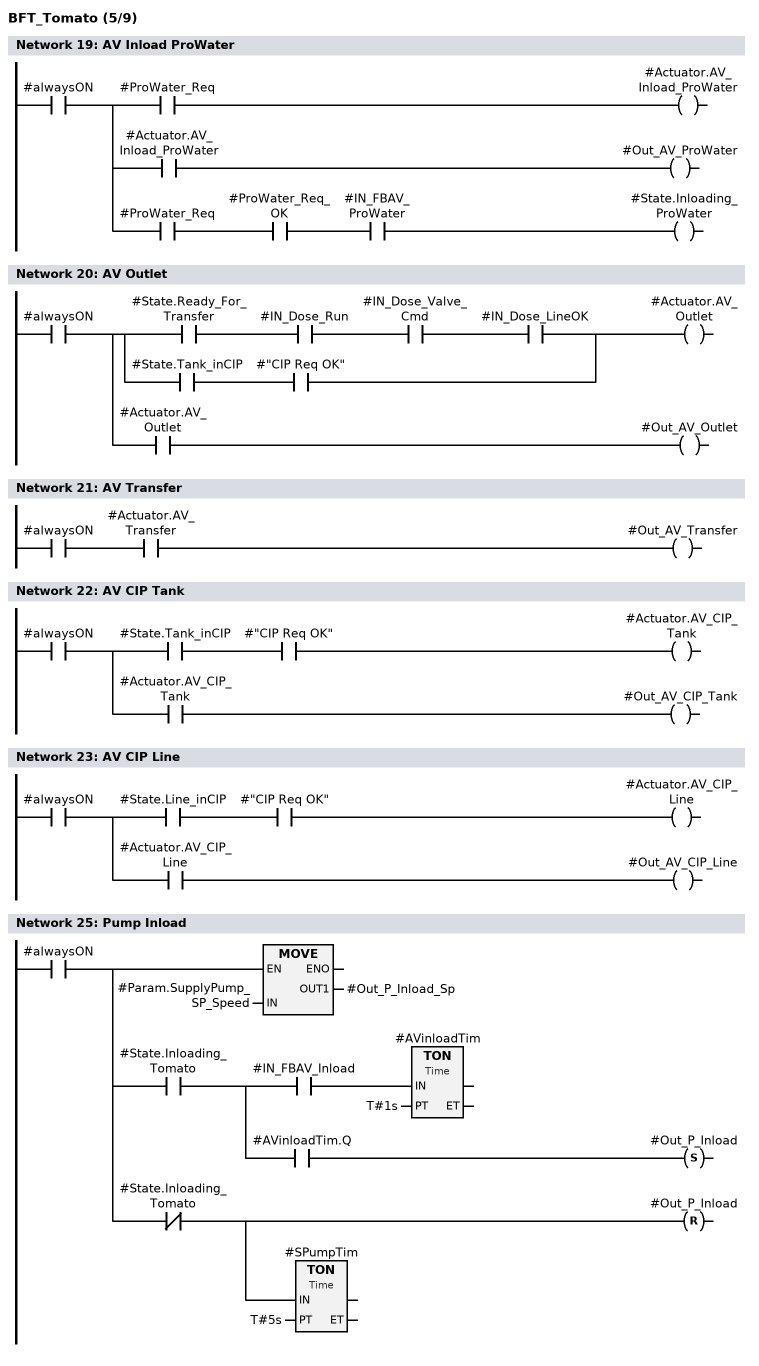
   RUNG wire#powerrail
      Contact( #alwaysON )
      wire#w1
      Contact( #ProWater_Req )
      Coil( #Actuator.AV_Inload_ProWater )
   END_RUNG
   RUNG wire#w1
      Contact( #Actuator.AV_Inload_ProWater )
      Coil( #Out_AV_ProWater )
   END_RUNG
   RUNG wire#w1
      Contact( #ProWater_Req )
      Contact( #ProWater_Req_OK )
      Contact( #IN_FBAV_ProWater )
      Coil( #State.Inloading_ProWater )
   END_RUNG
   // the same network as SCL:
   #Actuator.AV_Inload_ProWater := #alwaysON AND #ProWater_Req;
   #Out_AV_ProWater := #alwaysON AND #Actuator.AV_Inload_ProWater;
   #State.Inloading_ProWater := #alwaysON AND #ProWater_Req AND #ProWater_Req_OK AND #IN_FBAV_ProWater;
END_REGION

REGION Network 20: AV Outlet
   RUNG wire#powerrail
      Contact( #alwaysON )
      wire#w1
      Contact( #State.Ready_For_Transfer )
      Contact( #IN_Dose_Run )
      Contact( #IN_Dose_Valve_Cmd )
      Contact( #IN_Dose_LineOK )
      wire#w2
      Coil( #Actuator.AV_Outlet )
   END_RUNG
   RUNG wire#w1
      Contact( #State.Tank_inCIP )
      Contact( #"CIP Req OK" )
   END_RUNG wire#w2
   RUNG wire#w1
      Contact( #Actuator.AV_Outlet )
      Coil( #Out_AV_Outlet )
   END_RUNG
   // the same network as SCL:
   #Actuator.AV_Outlet := #alwaysON AND ((#State.Ready_For_Transfer AND #IN_Dose_Run AND #IN_Dose_Valve_Cmd AND #IN_Dose_LineOK) OR (#State.Tank_inCIP AND #"CIP Req OK"));
   #Out_AV_Outlet := #alwaysON AND #Actuator.AV_Outlet;
END_REGION

REGION Network 21: AV Transfer
   RUNG wire#powerrail
      Contact( #alwaysON )
      Contact( #Actuator.AV_Transfer )
      Coil( #Out_AV_Transfer )
   END_RUNG
   // the same network as SCL:
   #Out_AV_Transfer := #alwaysON AND #Actuator.AV_Transfer;
END_REGION

REGION Network 22: AV CIP Tank
   RUNG wire#powerrail
      Contact( #alwaysON )
      wire#w1
      Contact( #State.Tank_inCIP )
      Contact( #"CIP Req OK" )
      Coil( #Actuator.AV_CIP_Tank )
   END_RUNG
   RUNG wire#w1
      Contact( #Actuator.AV_CIP_Tank )
      Coil( #Out_AV_CIP_Tank )
   END_RUNG
   // the same network as SCL:
   #Actuator.AV_CIP_Tank := #alwaysON AND #State.Tank_inCIP AND #"CIP Req OK";
   #Out_AV_CIP_Tank := #alwaysON AND #Actuator.AV_CIP_Tank;
END_REGION

REGION Network 23: AV CIP Line
   RUNG wire#powerrail
      Contact( #alwaysON )
      wire#w1
      Contact( #State.Line_inCIP )
      Contact( #"CIP Req OK" )
      Coil( #Actuator.AV_CIP_Line )
   END_RUNG
   RUNG wire#w1
      Contact( #Actuator.AV_CIP_Line )
      Coil( #Out_AV_CIP_Line )
   END_RUNG
   // the same network as SCL:
   #Actuator.AV_CIP_Line := #alwaysON AND #State.Line_inCIP AND #"CIP Req OK";
   #Out_AV_CIP_Line := #alwaysON AND #Actuator.AV_CIP_Line;
END_REGION

REGION Network 25: Pump Inload
   RUNG wire#powerrail
      Contact( #alwaysON )
      wire#w1
      Move(in := #Param.SupplyPump_SP_Speed, out1 => #Out_P_Inload_Sp)
   END_RUNG
   RUNG wire#w1
      Contact( #State.Inloading_Tomato )
      wire#w2
      Contact( #IN_FBAV_Inload )
      { S7_Templates := "time_type := Time" } #AVinloadTim.TON(pt := T#1s, et =>)
   END_RUNG
   RUNG wire#w2
      Contact( #AVinloadTim.Q )
      S_Coil( #Out_P_Inload )
   END_RUNG
   RUNG wire#w1
      I_Contact( #State.Inloading_Tomato )
      wire#w3
      R_Coil( #Out_P_Inload )
   END_RUNG
   RUNG wire#w3
      { S7_Templates := "time_type := Time" } #SPumpTim.TON(pt := T#5s, et =>)
   END_RUNG
   // the same network as SCL:
   IF #alwaysON THEN #Out_P_Inload_Sp := #Param.SupplyPump_SP_Speed; END_IF;
   #_w1 := #alwaysON AND #State.Inloading_Tomato;
   #AVinloadTim(IN := #_w1 AND #IN_FBAV_Inload, PT := T#1s);   // TON
   IF #_w1 AND #AVinloadTim.Q THEN #Out_P_Inload := TRUE; END_IF;
   #_w2 := #alwaysON AND NOT #State.Inloading_Tomato;
   IF #_w2 THEN #Out_P_Inload := FALSE; END_IF;
   #SPumpTim(IN := #_w2, PT := T#5s);   // TON
END_REGION

REGION Network 26: Pump Transfer
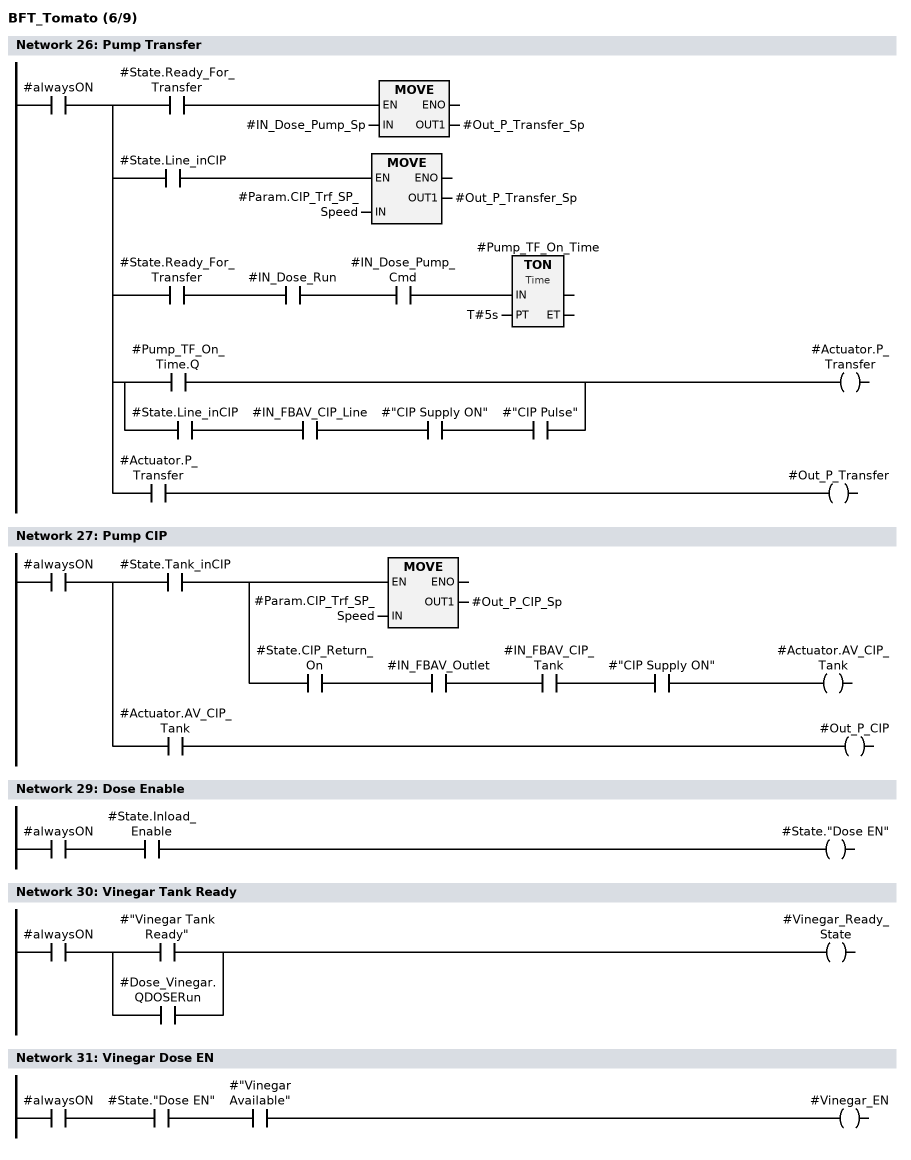
   RUNG wire#powerrail
      Contact( #alwaysON )
      wire#w1
      Contact( #State.Ready_For_Transfer )
      Move(in := #IN_Dose_Pump_Sp, out1 => #Out_P_Transfer_Sp)
   END_RUNG
   RUNG wire#w1
      Contact( #State.Line_inCIP )
      Move(in := #Param.CIP_Trf_SP_Speed, out1 => #Out_P_Transfer_Sp)
   END_RUNG
   RUNG wire#w1
      Contact( #State.Ready_For_Transfer )
      Contact( #IN_Dose_Run )
      Contact( #IN_Dose_Pump_Cmd )
      { S7_Templates := "time_type := Time" } #Pump_TF_On_Time.TON(pt := T#5s, et =>)
   END_RUNG
   RUNG wire#w1
      Contact( #Pump_TF_On_Time.Q )
      wire#w2
      Coil( #Actuator.P_Transfer )
   END_RUNG
   RUNG wire#w1
      Contact( #State.Line_inCIP )
      Contact( #IN_FBAV_CIP_Line )
      Contact( #"CIP Supply ON" )
      Contact( #"CIP Pulse" )
   END_RUNG wire#w2
   RUNG wire#w1
      Contact( #Actuator.P_Transfer )
      Coil( #Out_P_Transfer )
   END_RUNG
   // the same network as SCL:
   IF #alwaysON AND #State.Ready_For_Transfer THEN #Out_P_Transfer_Sp := #IN_Dose_Pump_Sp; END_IF;
   IF #alwaysON AND #State.Line_inCIP THEN #Out_P_Transfer_Sp := #Param.CIP_Trf_SP_Speed; END_IF;
   #Pump_TF_On_Time(IN := #alwaysON AND #State.Ready_For_Transfer AND #IN_Dose_Run AND #IN_Dose_Pump_Cmd,   // TON
                    PT := T#5s);
   #Actuator.P_Transfer := #alwaysON AND (#Pump_TF_On_Time.Q OR (#State.Line_inCIP AND #IN_FBAV_CIP_Line AND #"CIP Supply ON" AND #"CIP Pulse"));
   #Out_P_Transfer := #alwaysON AND #Actuator.P_Transfer;
END_REGION

REGION Network 27: Pump CIP
   RUNG wire#powerrail
      Contact( #alwaysON )
      wire#w1
      Contact( #State.Tank_inCIP )
      wire#w2
      Move(in := #Param.CIP_Trf_SP_Speed, out1 => #Out_P_CIP_Sp)
   END_RUNG
   RUNG wire#w2
      Contact( #State.CIP_Return_On )
      Contact( #IN_FBAV_Outlet )
      Contact( #IN_FBAV_CIP_Tank )
      Contact( #"CIP Supply ON" )
      Coil( #Actuator.AV_CIP_Tank )
   END_RUNG
   RUNG wire#w1
      Contact( #Actuator.AV_CIP_Tank )
      Coil( #Out_P_CIP )
   END_RUNG
   // the same network as SCL:
   #_w1 := #alwaysON AND #State.Tank_inCIP;
   IF #_w1 THEN #Out_P_CIP_Sp := #Param.CIP_Trf_SP_Speed; END_IF;
   #Actuator.AV_CIP_Tank := #_w1 AND #State.CIP_Return_On AND #IN_FBAV_Outlet AND #IN_FBAV_CIP_Tank AND #"CIP Supply ON";
   #Out_P_CIP := #alwaysON AND #Actuator.AV_CIP_Tank;
END_REGION

REGION Network 29: Dose Enable
   RUNG wire#powerrail
      Contact( #alwaysON )
      Contact( #State.Inload_Enable )
      Coil( #State."Dose EN" )
   END_RUNG
   // the same network as SCL:
   #State."Dose EN" := #alwaysON AND #State.Inload_Enable;
END_REGION

REGION Network 30: Vinegar Tank Ready
   RUNG wire#powerrail
      Contact( #alwaysON )
      wire#w1
      Contact( #"Vinegar Tank Ready" )
      wire#w2
      Coil( #Vinegar_Ready_State )
   END_RUNG
   RUNG wire#w1
      Contact( #Dose_Vinegar.QDOSERun )
   END_RUNG wire#w2
   // the same network as SCL:
   #Vinegar_Ready_State := #alwaysON AND (#"Vinegar Tank Ready" OR #Dose_Vinegar.QDOSERun);
END_REGION

REGION Network 31: Vinegar Dose EN
   RUNG wire#powerrail
      Contact( #alwaysON )
      Contact( #State."Dose EN" )
      Contact( #"Vinegar Available" )
      Coil( #Vinegar_EN )
   END_RUNG
   // the same network as SCL:
   #Vinegar_EN := #alwaysON AND #State."Dose EN" AND #"Vinegar Available";
END_REGION

REGION Network 32: Vinegar Setpoint
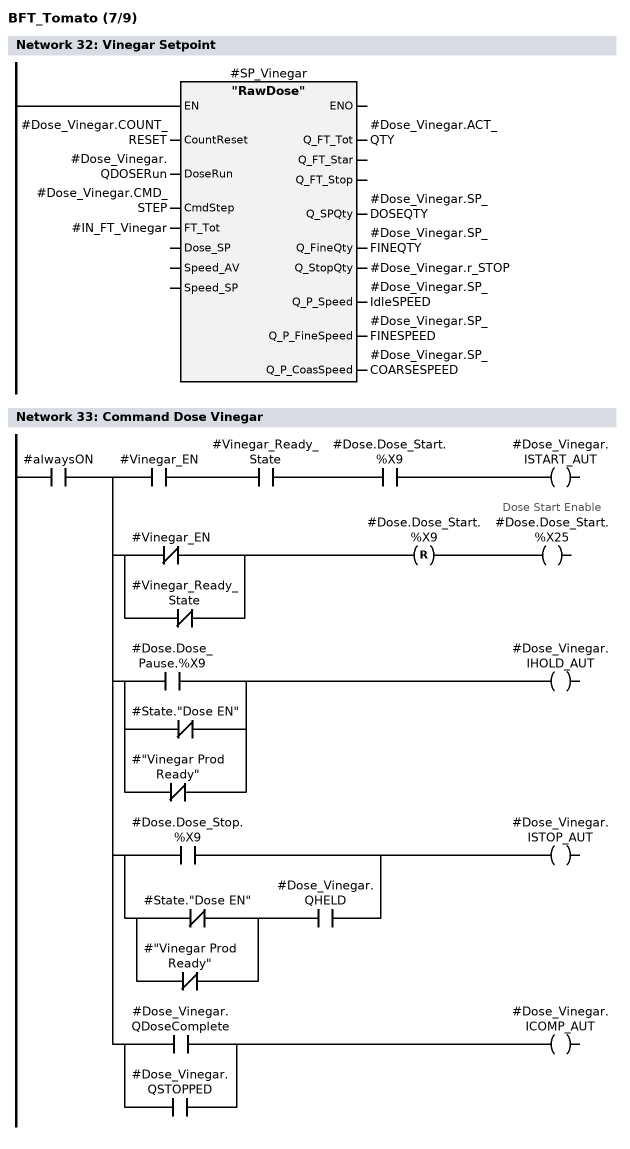
   RUNG wire#powerrail
      #SP_Vinegar(CountReset := #Dose_Vinegar.COUNT_RESET, DoseRun := #Dose_Vinegar.QDOSERun, CmdStep := #Dose_Vinegar.CMD_STEP, FT_Tot := #IN_FT_Vinegar, Dose_SP :=, Speed_AV :=, Speed_SP :=, Q_FT_Tot => #Dose_Vinegar.ACT_QTY, Q_FT_Star =>, Q_FT_Stop =>, Q_SPQty => #Dose_Vinegar.SP_DOSEQTY, Q_FineQty => #Dose_Vinegar.SP_FINEQTY, Q_StopQty => #Dose_Vinegar.r_STOP, Q_P_Speed => #Dose_Vinegar.SP_IdleSPEED, Q_P_FineSpeed => #Dose_Vinegar.SP_FINESPEED, Q_P_CoasSpeed => #Dose_Vinegar.SP_COARSESPEED)
   END_RUNG
   // the same network as SCL:
   #SP_Vinegar(CountReset := #Dose_Vinegar.COUNT_RESET,   // "RawDose"
               DoseRun := #Dose_Vinegar.QDOSERun,
               CmdStep := #Dose_Vinegar.CMD_STEP,
               FT_Tot := #IN_FT_Vinegar,
               Q_FT_Tot => #Dose_Vinegar.ACT_QTY,
               Q_SPQty => #Dose_Vinegar.SP_DOSEQTY,
               Q_FineQty => #Dose_Vinegar.SP_FINEQTY,
               Q_StopQty => #Dose_Vinegar.r_STOP,
               Q_P_Speed => #Dose_Vinegar.SP_IdleSPEED,
               Q_P_FineSpeed => #Dose_Vinegar.SP_FINESPEED,
               Q_P_CoasSpeed => #Dose_Vinegar.SP_COARSESPEED);
END_REGION

REGION Network 33: Command Dose Vinegar
   RUNG wire#powerrail
      Contact( #alwaysON )
      wire#w1
      Contact( #Vinegar_EN )
      Contact( #Vinegar_Ready_State )
      Contact( #Dose.Dose_Start.%X9 )
      Coil( #Dose_Vinegar.ISTART_AUT )
   END_RUNG
   RUNG wire#w1
      I_Contact( #Vinegar_EN )
      wire#w2
      R_Coil( #Dose.Dose_Start.%X9 )
      Coil( #Dose.Dose_Start.%X25 )   // Dose Start Enable
   END_RUNG
   RUNG wire#w1
      I_Contact( #Vinegar_Ready_State )
   END_RUNG wire#w2
   RUNG wire#w1
      Contact( #Dose.Dose_Pause.%X9 )
      wire#w3
      Coil( #Dose_Vinegar.IHOLD_AUT )
   END_RUNG
   RUNG wire#w1
      I_Contact( #State."Dose EN" )
   END_RUNG wire#w3
   RUNG wire#w1
      I_Contact( #"Vinegar Prod Ready" )
   END_RUNG wire#w3
   RUNG wire#w1
      Contact( #Dose.Dose_Stop.%X9 )
      wire#w4
      Coil( #Dose_Vinegar.ISTOP_AUT )
   END_RUNG
   RUNG wire#w1
      I_Contact( #State."Dose EN" )
      wire#w5
      Contact( #Dose_Vinegar.QHELD )
   END_RUNG wire#w4
   RUNG wire#w1
      I_Contact( #"Vinegar Prod Ready" )
   END_RUNG wire#w5
   RUNG wire#w1
      Contact( #Dose_Vinegar.QDoseComplete )
      wire#w6
      Coil( #Dose_Vinegar.ICOMP_AUT )
   END_RUNG
   RUNG wire#w1
      Contact( #Dose_Vinegar.QSTOPPED )
   END_RUNG wire#w6
   // the same network as SCL:
   #Dose_Vinegar.ISTART_AUT := #alwaysON AND #Vinegar_EN AND #Vinegar_Ready_State AND #Dose.Dose_Start.%X9;
   #_w1 := #alwaysON AND (NOT #Vinegar_EN OR NOT #Vinegar_Ready_State);
   IF #_w1 THEN #Dose.Dose_Start.%X9 := FALSE; END_IF;
   #Dose.Dose_Start.%X25 := #_w1;   // Dose Start Enable
   #Dose_Vinegar.IHOLD_AUT := #alwaysON AND (#Dose.Dose_Pause.%X9 OR NOT #State."Dose EN" OR NOT #"Vinegar Prod Ready");
   #Dose_Vinegar.ISTOP_AUT := #alwaysON AND (#Dose.Dose_Stop.%X9 OR ((NOT #State."Dose EN" OR NOT #"Vinegar Prod Ready") AND #Dose_Vinegar.QHELD));
   #Dose_Vinegar.ICOMP_AUT := #alwaysON AND (#Dose_Vinegar.QDoseComplete OR #Dose_Vinegar.QSTOPPED);
END_REGION

REGION Network 34: Dose Vinegar
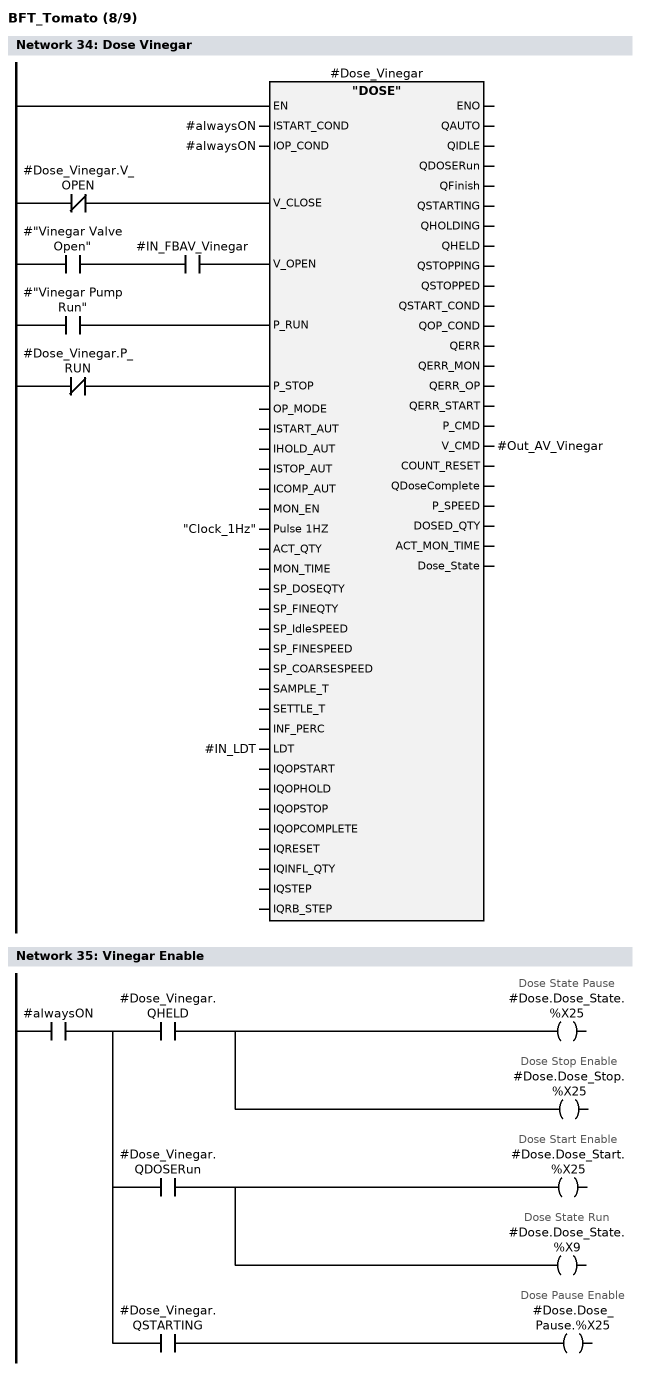
   RUNG wire#powerrail
      #Dose_Vinegar(V_CLOSE := wire#w1, V_OPEN := wire#w2, P_RUN := wire#w3, P_STOP := wire#w4, ISTART_COND := #alwaysON, IOP_COND := #alwaysON, OP_MODE :=, ISTART_AUT :=, IHOLD_AUT :=, ISTOP_AUT :=, ICOMP_AUT :=, MON_EN :=, "Pulse 1HZ" := "Clock_1Hz", ACT_QTY :=, MON_TIME :=, SP_DOSEQTY :=, SP_FINEQTY :=, SP_IdleSPEED :=, SP_FINESPEED :=, SP_COARSESPEED :=, SAMPLE_T :=, SETTLE_T :=, INF_PERC :=, LDT := #IN_LDT, IQOPSTART :=, IQOPHOLD :=, IQOPSTOP :=, IQOPCOMPLETE :=, IQRESET :=, IQINFL_QTY :=, IQSTEP :=, IQRB_STEP :=, QAUTO =>, QIDLE =>, QDOSERun =>, QFinish =>, QSTARTING =>, QHOLDING =>, QHELD =>, QSTOPPING =>, QSTOPPED =>, QSTART_COND =>, QOP_COND =>, QERR =>, QERR_MON =>, QERR_OP =>, QERR_START =>, P_CMD =>, V_CMD => #Out_AV_Vinegar, COUNT_RESET =>, QDoseComplete =>, P_SPEED =>, DOSED_QTY =>, ACT_MON_TIME =>, Dose_State =>)
   END_RUNG
   RUNG wire#powerrail
      I_Contact( #Dose_Vinegar.V_OPEN )
   END_RUNG wire#w1
   RUNG wire#powerrail
      Contact( #"Vinegar Valve Open" )
      Contact( #IN_FBAV_Vinegar )
   END_RUNG wire#w2
   RUNG wire#powerrail
      Contact( #"Vinegar Pump Run" )
   END_RUNG wire#w3
   RUNG wire#powerrail
      I_Contact( #Dose_Vinegar.P_RUN )
   END_RUNG wire#w4
   // the same network as SCL:
   #Dose_Vinegar(ISTART_COND := #alwaysON,   // "DOSE"
                 IOP_COND := #alwaysON,
                 V_CLOSE := NOT #Dose_Vinegar.V_OPEN,
                 V_OPEN := #"Vinegar Valve Open" AND #IN_FBAV_Vinegar,
                 P_RUN := #"Vinegar Pump Run",
                 P_STOP := NOT #Dose_Vinegar.P_RUN,
                 "Pulse 1HZ" := "Clock_1Hz",
                 LDT := #IN_LDT,
                 V_CMD => #Out_AV_Vinegar);
END_REGION

REGION Network 35: Vinegar Enable
   RUNG wire#powerrail
      Contact( #alwaysON )
      wire#w1
      Contact( #Dose_Vinegar.QHELD )
      wire#w2
      Coil( #Dose.Dose_State.%X25 )   // Dose State Pause
   END_RUNG
   RUNG wire#w2
      Coil( #Dose.Dose_Stop.%X25 )   // Dose Stop Enable
   END_RUNG
   RUNG wire#w1
      Contact( #Dose_Vinegar.QDOSERun )
      wire#w3
      Coil( #Dose.Dose_Start.%X25 )   // Dose Start Enable
   END_RUNG
   RUNG wire#w3
      Coil( #Dose.Dose_State.%X9 )   // Dose State Run
   END_RUNG
   RUNG wire#w1
      Contact( #Dose_Vinegar.QSTARTING )
      Coil( #Dose.Dose_Pause.%X25 )   // Dose Pause Enable
   END_RUNG
   // the same network as SCL:
   #Dose.Dose_State.%X25 := #alwaysON AND #Dose_Vinegar.QHELD;   // Dose State Pause
   #Dose.Dose_Stop.%X25 := #Dose.Dose_State.%X25;   // Dose Stop Enable
   #Dose.Dose_Start.%X25 := #alwaysON AND #Dose_Vinegar.QDOSERun;   // Dose Start Enable
   #Dose.Dose_State.%X9 := #Dose.Dose_Start.%X25;   // Dose State Run
   #Dose.Dose_Pause.%X25 := #alwaysON AND #Dose_Vinegar.QSTARTING;   // Dose Pause Enable
END_REGION

REGION Network 36: Vinegar Header Req
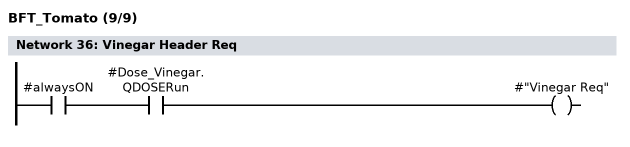
   RUNG wire#powerrail
      Contact( #alwaysON )
      Contact( #Dose_Vinegar.QDOSERun )
      Coil( #"Vinegar Req" )
   END_RUNG
   // the same network as SCL:
   #"Vinegar Req" := #alwaysON AND #Dose_Vinegar.QDOSERun;
END_REGION
END_FUNCTION_BLOCK

FUNCTION_BLOCK "RawDose"   // FB103, LAD
{ S7_Optimized_Access := 'TRUE' }
VERSION : 0.1
// stored: AutoNumber false, IsIECCheckEnabled false, IsRetainMemResEnabled false, MemoryReserve 100, SetENOAutomatically false, UDAEnableTagReadback false
   VAR_INPUT
      CountReset : Bool;
      DoseRun : Bool;
      CmdStep : Int;
      FT_Tot : Real;
      Dose_SP : Real;
      Speed_AV : Real;
      Speed_SP : Real;
   END_VAR
   VAR_OUTPUT
      Q_FT_Tot : Real;
      Q_FT_Star : Real;
      Q_FT_Stop : Real;
      Q_SPQty : Real;
      Q_FineQty : Real;
      Q_StopQty : Real;
      Q_P_Speed : Real;
      Q_P_FineSpeed : Real;
      Q_P_CoasSpeed : Real;
   END_VAR
   VAR RETAIN
      Para : Struct
         "SP_Qty_Stop%" : Real := 3.0;
         "SP_Qty_Fine%" : Real := 20.0;
         SP_Qty_Stop : Real;
         SP_Qty_Fine : Real;
         SP_Pump_Co : Real := 80.0;
         SP_Pump_Fi : Real := 20.0;
      END_STRUCT;
   END_VAR
   VAR
      alwaysON { S7_SetPoint := 'True'} : Bool;
      DosePE : Bool;
   END_VAR
   VAR_TEMP   // added for the SCL form of the ladder/FBD networks
      _w1 : Bool;
      _w2 : Bool;
      _w3 : Bool;
   END_VAR
BEGIN

REGION Network 1: alwaysON
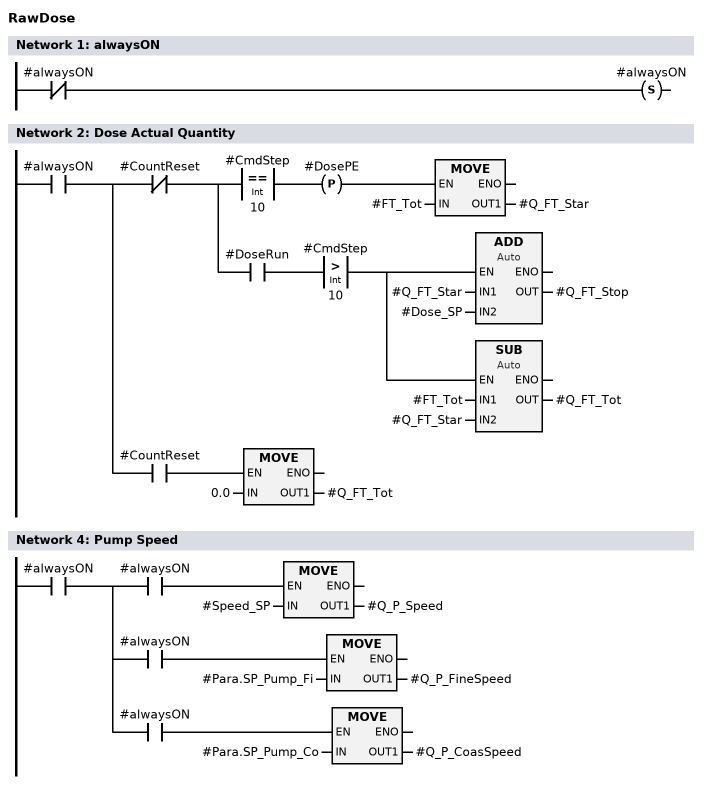
   RUNG wire#powerrail
      I_Contact( #alwaysON )
      S_Coil( #alwaysON )
   END_RUNG
   // the same network as SCL:
   IF NOT #alwaysON THEN #alwaysON := TRUE; END_IF;
END_REGION

REGION Network 2: Dose Actual Quantity
   RUNG wire#powerrail
      Contact( #alwaysON )
      wire#w1
      I_Contact( #CountReset )
      wire#w2
      { S7_Templates := "SrcType := Int" } EQ_Contact(in1 := #CmdStep, in2 := 10)
      P_Trig( #DosePE )
      Move(in := #FT_Tot, out1 => #Q_FT_Star)
   END_RUNG
   RUNG wire#w2
      Contact( #DoseRun )
      { S7_Templates := "SrcType := Int" } GT_Contact(in1 := #CmdStep, in2 := 10)
      wire#w3
      Add(in1 := #Q_FT_Star, in2 := #Dose_SP, out => #Q_FT_Stop)
   END_RUNG
   RUNG wire#w3
      Sub(in1 := #FT_Tot, in2 := #Q_FT_Star, out => #Q_FT_Tot)
   END_RUNG
   RUNG wire#w1
      Contact( #CountReset )
      Move(in := 0.0, out1 => #Q_FT_Tot)
   END_RUNG
   // the same network as SCL:
   #_w1 := #alwaysON AND NOT #CountReset;
   #_w2 := #_w1 AND (#CmdStep = 10);
   #_w3 := #_w2 AND NOT #DosePE;   // rising edge
   #DosePE := #_w2;
   IF #_w3 THEN #Q_FT_Star := #FT_Tot; END_IF;
   IF #_w1 AND #DoseRun AND (#CmdStep > 10) THEN
       #Q_FT_Stop := #Q_FT_Star + #Dose_SP;
       #Q_FT_Tot := #FT_Tot - #Q_FT_Star;
   END_IF;
   IF #alwaysON AND #CountReset THEN #Q_FT_Tot := 0.0; END_IF;
END_REGION

NETWORK
TITLE = Quantity Calculation
// SP Quantity
      L     #Dose_SP;
      T     #Q_SPQty;
// Fine Quantity Calculation
      L     #Dose_SP;
      L     #Para."SP_Qty_Fine%";
      *R;
      L     100.0;
      /R;
      T     #Para.SP_Qty_Fine;

      L     #Dose_SP;
      L     #Para.SP_Qty_Fine;
      -R;
      T     #Q_FineQty;

// Stop Quantity Calculation
      L     #Dose_SP;
      L     #Para."SP_Qty_Stop%";
      *R;
      L     100.0;
      /R;
      T     #Para.SP_Qty_Stop;

      L     #Dose_SP;
      L     #Para.SP_Qty_Stop;
      -R;
      T     #Q_StopQty;


REGION Network 4: Pump Speed
   RUNG wire#powerrail
      Contact( #alwaysON )
      wire#w1
      Contact( #alwaysON )
      Move(in := #Speed_SP, out1 => #Q_P_Speed)
   END_RUNG
   RUNG wire#w1
      Contact( #alwaysON )
      Move(in := #Para.SP_Pump_Fi, out1 => #Q_P_FineSpeed)
   END_RUNG
   RUNG wire#w1
      Contact( #alwaysON )
      Move(in := #Para.SP_Pump_Co, out1 => #Q_P_CoasSpeed)
   END_RUNG
   // the same network as SCL:
   IF #alwaysON AND #alwaysON THEN
       #Q_P_Speed := #Speed_SP;
       #Q_P_FineSpeed := #Para.SP_Pump_Fi;
       #Q_P_CoasSpeed := #Para.SP_Pump_Co;
   END_IF;
END_REGION
END_FUNCTION_BLOCK

FUNCTION_BLOCK "DOSE"   // FB102, LAD
TITLE = Dosing Module type 1; 1 adustable speed pump and 1 auto valve.
{ S7_Optimized_Access := 'FALSE' }
AUTHOR : N@wi
FAMILY : DOSE
NAME : DOSE
VERSION : 0.1
// Dosing Module type 1:
// Use for Dosing module with adjustable speed pump and auto valve. Coarse dosing 
// and Fine dosing by adjusting the pump speed.
// stored: AutoNumber false, IsIECCheckEnabled false, SetENOAutomatically false, UDAEnableTagReadback false
   VAR_INPUT
      ISTART_COND : Bool;   // Starting Condition. 1 = Dose sequence can be Start
      IOP_COND : Bool;   // Operating Condition. 0 = Dose will be hold
      V_CLOSE : Bool;   // Valve in close position
      V_OPEN : Bool;   // Valve in open position
      P_RUN : Bool;   // Pump Run
      P_STOP : Bool;   // Pump Stop
      OP_MODE : Bool := TRUE;   // Dosing Mode; 0 = MANUAL; 1 = AUTO
      ISTART_AUT : Bool;   // Start command in Auto dosing mode
      IHOLD_AUT : Bool;   // Hold command in Auto dosing mode
      ISTOP_AUT : Bool;   // Stop command in Auto dosing mode
      ICOMP_AUT : Bool;   // Complete command in Auto dosing mode
      MON_EN : Bool;   // Monitoring time enable
      "Pulse 1HZ" : Bool;
      ACT_QTY : Real;   // Actual Counter quantity
      MON_TIME : Real := 60.0;   // Monitoring Time (in second)
      SP_DOSEQTY : Real;   // Dosing Setpoint Quantity
      SP_FINEQTY : Real;   // Fine Quantity Setpoint
      SP_IdleSPEED : Real;
      SP_FINESPEED : Real;   // Fine Speed Setpoint
      SP_COARSESPEED : Real;   // Coarse Speed Setpoint
      SAMPLE_T : Real := 1.0;   // Sample Time
      SETTLE_T : Real := 3.0;   // Settling Time
      INF_PERC : Real := 2.0;   // Percentage of calculated infligh qty (in %)
      LDT : Date_And_Time;
   END_VAR
   VAR_OUTPUT
      QAUTO : Bool;   // Selected Operation Mode 0 = MANUAL; 1 = AUTO
      QIDLE : Bool;   // Dosing module in IDLE state
      QDOSERun : Bool;   // Dosing module in Running state
      QFinish : Bool;   // Dosing module in Finish
      QSTARTING : Bool;   // Dosing module in STARTING state
      QHOLDING : Bool;   // Dosing module in HOLDING state
      QHELD : Bool;   // Dosing module in HELD state
      QSTOPPING : Bool;   // Dosing module in STOPPING state
      QSTOPPED : Bool;   // Dosing module in STOPPED state
      QSTART_COND : Bool;   // Starting Condition are met
      QOP_COND : Bool;   // Operating Condition are met
      QERR : Bool;   // General Error
      QERR_MON : Bool;   // Error cause by runtime monitoring error
      QERR_OP : Bool;   // Error cause by operating condition not OK
      QERR_START : Bool;   // Error cause by start condition not OK
      P_CMD : Bool;   // Pump Start command
      V_CMD : Bool;   // Valve Open command
      COUNT_RESET : Bool;   // Counter reset command
      QDoseComplete : Bool;
      P_SPEED : Real;   // Pump speed setpoint
      DOSED_QTY : Real;   // Dosed quantity
      ACT_MON_TIME : Real;   // Actual Monitoring Time
      Dose_State : Word;
   END_VAR
   VAR_IN_OUT
      IQOPSTART : Bool;   // Start command by operator in Manual dosing mode
      IQOPHOLD : Bool;   // Hold command by operator in Manual dosing mode
      IQOPSTOP : Bool;   // Stop command by operator in Manual dosing mode
      IQOPCOMPLETE : Bool;   // Complete command by operator in Manual dosing mode
      IQRESET : Bool;   // Reset Error
      IQINFL_QTY : Real := 3.0e+0;   // Inflight quantity. Will be calculated in end of dosing for the next dosing.
      IQSTEP : Int;   // Actual step
      IQRB_STEP : Int;   // Roll Back Step
   END_VAR
   VAR DB_SPECIFIC
      b_IDLE : Bool;   // Dosing module in IDLE state
      b_Finish : Bool;   // Dosing module in Finish state
      b_STARTING : Bool;   // Dosing module in STARTING state
      b_HOLDING : Bool;   // Dosing module in HOLDING state
      b_HELD : Bool;   // Dosing module in HELD state
      b_STOPPING : Bool;   // Dosing module in STOPPING state
      b_STOPPED : Bool;   // Dosing module in STOPPED state
      b_START : Bool;   // Start command
      b_HOLD : Bool;   // Hold command
      b_STOP : Bool;   // Stop command
      b_COMP : Bool;   // Complete command
      b_START_AP : Bool;   // Start command Auto Pulse
      b_HOLD_AP : Bool;   // Hold command Auto Pulse
      b_STOP_AP : Bool;   // Stop command Auto Pulse
      b_COMP_AP : Bool;   // Complete command Auto Pulse
      b_START_MP : Bool;   // Start command Manual Pulse
      b_HOLD_MP : Bool;   // Hold command Manual Pulse
      b_STOP_MP : Bool;   // Stop command Manual Pulse
      b_COMP_MP : Bool;   // Complete command Manual Pulse
      b_ERR_MON : Bool;   // Error cause by runtime monitoring error
      b_ERR_OP : Bool;   // Error cause by operating condition not OK
      b_ERR_START : Bool;   // Error cause by start condition not OK
      PE_Setle : Bool;
      PE_Mon : Bool;
      CMD_STEP : Int;   // STEP command
      r_MON : Real;   // Actual Monitoring Time
      r_STOP : Real;   // Quantity to stop dosing
      r_FINE : Real;   // Quantity change to fine dosing
      r_SETTLE_T : Real;   // Settling Time
      r_INFLIGHT : Real;   // Saved inflight qty
      r_DIFF : Real;   // Dosed Qty - SP Quantity
      r_INFDIFF : Real;   // Diff of Inflight qty to be added to new inflight
      r_INFPERC { ExternalAccessible := 'False'; ExternalVisible := 'False'; ExternalWritable := 'False'} : Real;
      LDT_Start { S7_SetPoint := 'True'} : Date_And_Time;
      LDT_Finish : Date_And_Time;
      TimeDose : Time;
      LastTimeDose : Time;
      PE_LDTStart : Bool;
      PE_LDTFinish : Bool;
      PE_LDTStore : Bool;
      PE_QtyStart : Bool;
      PE_QtyFinish : Bool;
      PE_QtyStore : Bool;
      AlwaysON : Bool;
      LastQtyDose : Real;
   END_VAR
   VAR_TEMP   // added for the SCL form of the ladder/FBD networks
      _w1 : Bool;
      _w2 : Bool;
      _w3 : Bool;
      _w4 : Bool;
   END_VAR
BEGIN

REGION Network 1: AlwaysON
   // Copying the command step number to actual step number to avoid double step in 
   // one scan.
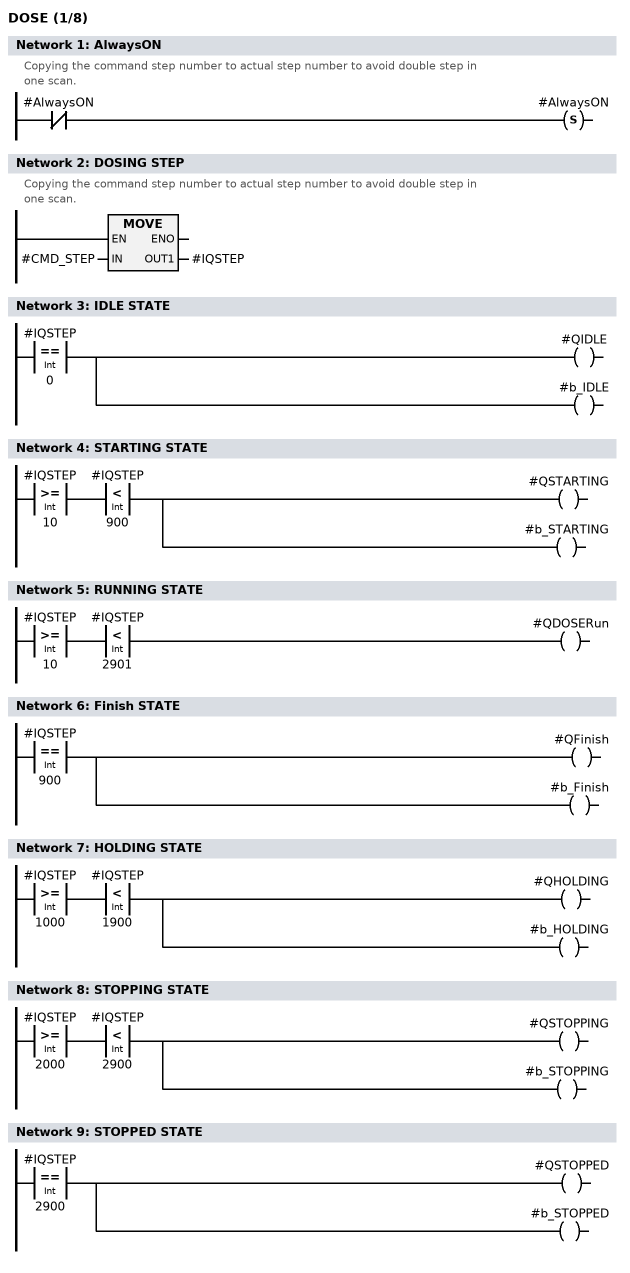
   RUNG wire#powerrail
      I_Contact( #AlwaysON )
      S_Coil( #AlwaysON )
   END_RUNG
   // the same network as SCL:
   IF NOT #AlwaysON THEN #AlwaysON := TRUE; END_IF;
END_REGION

REGION Network 2: DOSING STEP
   // Copying the command step number to actual step number to avoid double step in 
   // one scan.
   RUNG wire#powerrail
      { S7_GenerateENO := "TRUE" } Move(in := #CMD_STEP, out1 => #IQSTEP)
   END_RUNG
   // the same network as SCL:
   #IQSTEP := #CMD_STEP;
END_REGION

REGION Network 3: IDLE STATE
   RUNG wire#powerrail
      { S7_Templates := "SrcType := Int" } EQ_Contact(in1 := #IQSTEP, in2 := 0)
      wire#w1
      Coil( #QIDLE )
   END_RUNG
   RUNG wire#w1
      Coil( #b_IDLE )
   END_RUNG
   // the same network as SCL:
   #QIDLE := #IQSTEP = 0;
   #b_IDLE := #QIDLE;
END_REGION

REGION Network 4: STARTING STATE
   RUNG wire#powerrail
      { S7_Templates := "SrcType := Int" } GE_Contact(in1 := #IQSTEP, in2 := 10)
      { S7_Templates := "SrcType := Int" } LT_Contact(in1 := #IQSTEP, in2 := 900)
      wire#w1
      Coil( #QSTARTING )
   END_RUNG
   RUNG wire#w1
      Coil( #b_STARTING )
   END_RUNG
   // the same network as SCL:
   #QSTARTING := (#IQSTEP >= 10) AND (#IQSTEP < 900);
   #b_STARTING := #QSTARTING;
END_REGION

REGION Network 5: RUNNING STATE
   RUNG wire#powerrail
      { S7_Templates := "SrcType := Int" } GE_Contact(in1 := #IQSTEP, in2 := 10)
      { S7_Templates := "SrcType := Int" } LT_Contact(in1 := #IQSTEP, in2 := 2901)
      Coil( #QDOSERun )
   END_RUNG
   // the same network as SCL:
   #QDOSERun := (#IQSTEP >= 10) AND (#IQSTEP < 2901);
END_REGION

REGION Network 6: Finish STATE
   RUNG wire#powerrail
      { S7_Templates := "SrcType := Int" } EQ_Contact(in1 := #IQSTEP, in2 := 900)
      wire#w1
      Coil( #QFinish )
   END_RUNG
   RUNG wire#w1
      Coil( #b_Finish )
   END_RUNG
   // the same network as SCL:
   #QFinish := #IQSTEP = 900;
   #b_Finish := #QFinish;
END_REGION

REGION Network 7: HOLDING STATE
   RUNG wire#powerrail
      { S7_Templates := "SrcType := Int" } GE_Contact(in1 := #IQSTEP, in2 := 1000)
      { S7_Templates := "SrcType := Int" } LT_Contact(in1 := #IQSTEP, in2 := 1900)
      wire#w1
      Coil( #QHOLDING )
   END_RUNG
   RUNG wire#w1
      Coil( #b_HOLDING )
   END_RUNG
   // the same network as SCL:
   #QHOLDING := (#IQSTEP >= 1000) AND (#IQSTEP < 1900);
   #b_HOLDING := #QHOLDING;
END_REGION

REGION Network 8: STOPPING STATE
   RUNG wire#powerrail
      { S7_Templates := "SrcType := Int" } GE_Contact(in1 := #IQSTEP, in2 := 2000)
      { S7_Templates := "SrcType := Int" } LT_Contact(in1 := #IQSTEP, in2 := 2900)
      wire#w1
      Coil( #QSTOPPING )
   END_RUNG
   RUNG wire#w1
      Coil( #b_STOPPING )
   END_RUNG
   // the same network as SCL:
   #QSTOPPING := (#IQSTEP >= 2000) AND (#IQSTEP < 2900);
   #b_STOPPING := #QSTOPPING;
END_REGION

REGION Network 9: STOPPED STATE
   RUNG wire#powerrail
      { S7_Templates := "SrcType := Int" } EQ_Contact(in1 := #IQSTEP, in2 := 2900)
      wire#w1
      Coil( #QSTOPPED )
   END_RUNG
   RUNG wire#w1
      Coil( #b_STOPPED )
   END_RUNG
   // the same network as SCL:
   #QSTOPPED := #IQSTEP = 2900;
   #b_STOPPED := #QSTOPPED;
END_REGION

REGION Network 10: START COMMAND
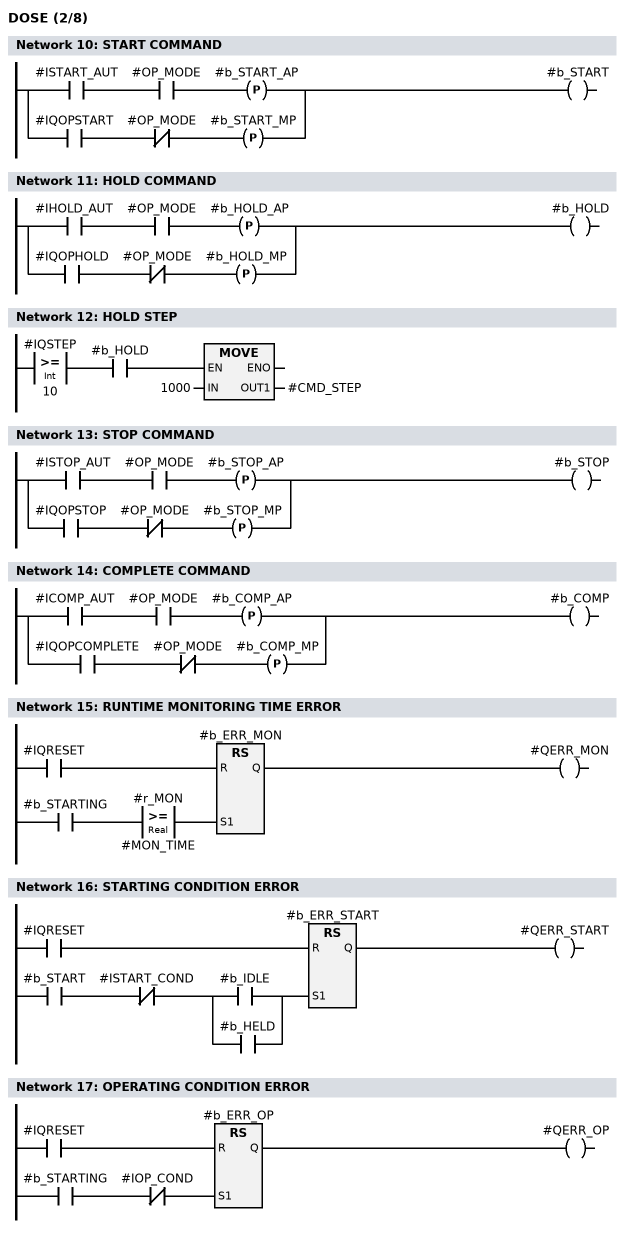
   RUNG wire#powerrail
      Contact( #ISTART_AUT )
      Contact( #OP_MODE )
      P_Trig( #b_START_AP )
      wire#w1
      Coil( #b_START )
   END_RUNG
   RUNG wire#powerrail
      Contact( #IQOPSTART )
      I_Contact( #OP_MODE )
      P_Trig( #b_START_MP )
   END_RUNG wire#w1
   // the same network as SCL:
   #_w1 := #ISTART_AUT AND #OP_MODE;
   #_w2 := #_w1 AND NOT #b_START_AP;   // rising edge
   #b_START_AP := #_w1;
   #_w3 := #IQOPSTART AND NOT #OP_MODE;
   #_w4 := #_w3 AND NOT #b_START_MP;   // rising edge
   #b_START_MP := #_w3;
   #b_START := #_w2 OR #_w4;
END_REGION

REGION Network 11: HOLD COMMAND
   RUNG wire#powerrail
      Contact( #IHOLD_AUT )
      Contact( #OP_MODE )
      P_Trig( #b_HOLD_AP )
      wire#w1
      Coil( #b_HOLD )
   END_RUNG
   RUNG wire#powerrail
      Contact( #IQOPHOLD )
      I_Contact( #OP_MODE )
      P_Trig( #b_HOLD_MP )
   END_RUNG wire#w1
   // the same network as SCL:
   #_w1 := #IHOLD_AUT AND #OP_MODE;
   #_w2 := #_w1 AND NOT #b_HOLD_AP;   // rising edge
   #b_HOLD_AP := #_w1;
   #_w3 := #IQOPHOLD AND NOT #OP_MODE;
   #_w4 := #_w3 AND NOT #b_HOLD_MP;   // rising edge
   #b_HOLD_MP := #_w3;
   #b_HOLD := #_w2 OR #_w4;
END_REGION

REGION Network 12: HOLD STEP
   RUNG wire#powerrail
      { S7_Templates := "SrcType := Int" } GE_Contact(in1 := #IQSTEP, in2 := 10)
      Contact( #b_HOLD )
      { S7_GenerateENO := "TRUE" } Move(in := 1000, out1 => #CMD_STEP)
   END_RUNG
   // the same network as SCL:
   IF (#IQSTEP >= 10) AND #b_HOLD THEN #CMD_STEP := 1000; END_IF;
END_REGION

REGION Network 13: STOP COMMAND
   RUNG wire#powerrail
      Contact( #ISTOP_AUT )
      Contact( #OP_MODE )
      P_Trig( #b_STOP_AP )
      wire#w1
      Coil( #b_STOP )
   END_RUNG
   RUNG wire#powerrail
      Contact( #IQOPSTOP )
      I_Contact( #OP_MODE )
      P_Trig( #b_STOP_MP )
   END_RUNG wire#w1
   // the same network as SCL:
   #_w1 := #ISTOP_AUT AND #OP_MODE;
   #_w2 := #_w1 AND NOT #b_STOP_AP;   // rising edge
   #b_STOP_AP := #_w1;
   #_w3 := #IQOPSTOP AND NOT #OP_MODE;
   #_w4 := #_w3 AND NOT #b_STOP_MP;   // rising edge
   #b_STOP_MP := #_w3;
   #b_STOP := #_w2 OR #_w4;
END_REGION

REGION Network 14: COMPLETE COMMAND
   RUNG wire#powerrail
      Contact( #ICOMP_AUT )
      Contact( #OP_MODE )
      P_Trig( #b_COMP_AP )
      wire#w1
      Coil( #b_COMP )
   END_RUNG
   RUNG wire#powerrail
      Contact( #IQOPCOMPLETE )
      I_Contact( #OP_MODE )
      P_Trig( #b_COMP_MP )
   END_RUNG wire#w1
   // the same network as SCL:
   #_w1 := #ICOMP_AUT AND #OP_MODE;
   #_w2 := #_w1 AND NOT #b_COMP_AP;   // rising edge
   #b_COMP_AP := #_w1;
   #_w3 := #IQOPCOMPLETE AND NOT #OP_MODE;
   #_w4 := #_w3 AND NOT #b_COMP_MP;   // rising edge
   #b_COMP_MP := #_w3;
   #b_COMP := #_w2 OR #_w4;
END_REGION

REGION Network 15: RUNTIME MONITORING TIME ERROR
   RUNG wire#powerrail
      Contact( #IQRESET )
      S_RS(operand := #b_ERR_MON, s1 := wire#w1)
      Coil( #QERR_MON )
   END_RUNG
   RUNG wire#powerrail
      Contact( #b_STARTING )
      { S7_Templates := "SrcType := Real" } GE_Contact(in1 := #r_MON, in2 := #MON_TIME)
   END_RUNG wire#w1
   // the same network as SCL:
   IF #IQRESET THEN
       #b_ERR_MON := FALSE;   // RS flip-flop
   END_IF;
   IF #b_STARTING AND (#r_MON >= #MON_TIME) THEN #b_ERR_MON := TRUE; END_IF;
   #QERR_MON := #b_ERR_MON;
END_REGION

REGION Network 16: STARTING CONDITION ERROR
   RUNG wire#powerrail
      Contact( #IQRESET )
      S_RS(operand := #b_ERR_START, s1 := wire#w2)
      Coil( #QERR_START )
   END_RUNG
   RUNG wire#powerrail
      Contact( #b_START )
      I_Contact( #ISTART_COND )
      wire#w1
      Contact( #b_IDLE )
   END_RUNG wire#w2
   RUNG wire#w1
      Contact( #b_HELD )
   END_RUNG wire#w2
   // the same network as SCL:
   IF #IQRESET THEN
       #b_ERR_START := FALSE;   // RS flip-flop
   END_IF;
   IF #b_START AND NOT #ISTART_COND AND (#b_IDLE OR #b_HELD) THEN #b_ERR_START := TRUE; END_IF;
   #QERR_START := #b_ERR_START;
END_REGION

REGION Network 17: OPERATING CONDITION ERROR
   RUNG wire#powerrail
      Contact( #IQRESET )
      S_RS(operand := #b_ERR_OP, s1 := wire#w1)
      Coil( #QERR_OP )
   END_RUNG
   RUNG wire#powerrail
      Contact( #b_STARTING )
      I_Contact( #IOP_COND )
   END_RUNG wire#w1
   // the same network as SCL:
   IF #IQRESET THEN
       #b_ERR_OP := FALSE;   // RS flip-flop
   END_IF;
   IF #b_STARTING AND NOT #IOP_COND THEN #b_ERR_OP := TRUE; END_IF;
   #QERR_OP := #b_ERR_OP;
END_REGION

REGION Network 18: GENERAL ERROR
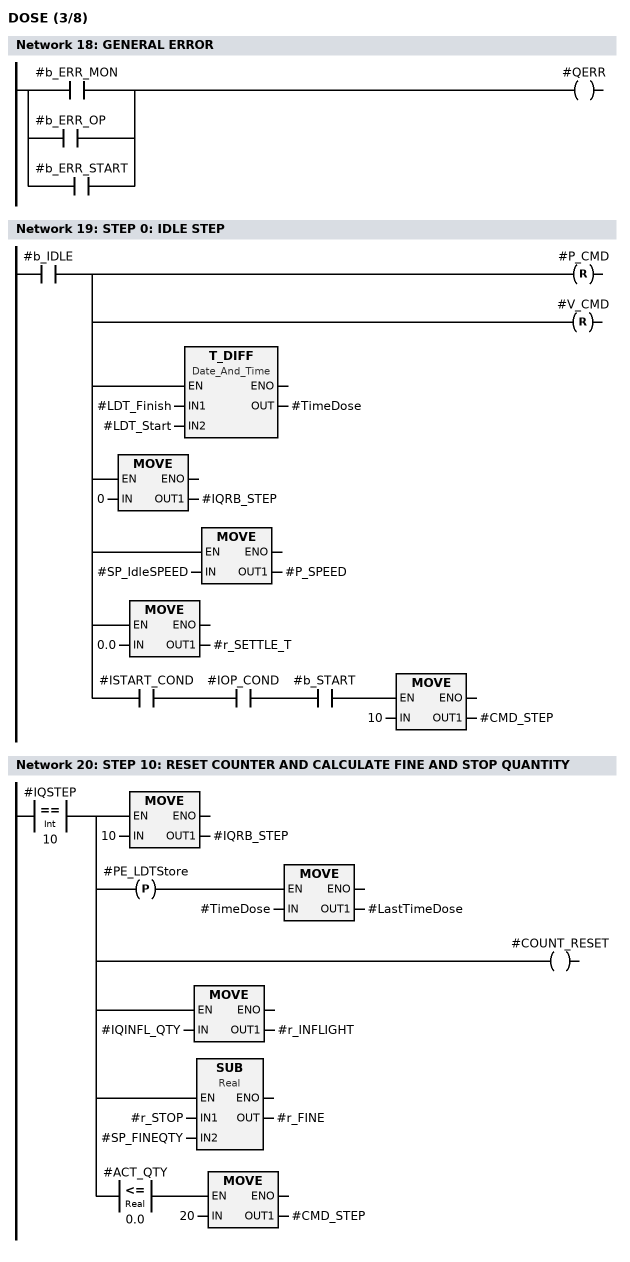
   RUNG wire#powerrail
      Contact( #b_ERR_MON )
      wire#w1
      Coil( #QERR )
   END_RUNG
   RUNG wire#powerrail
      Contact( #b_ERR_OP )
   END_RUNG wire#w1
   RUNG wire#powerrail
      Contact( #b_ERR_START )
   END_RUNG wire#w1
   // the same network as SCL:
   #QERR := #b_ERR_MON OR #b_ERR_OP OR #b_ERR_START;
END_REGION

REGION Network 19: STEP 0: IDLE STEP
   RUNG wire#powerrail
      Contact( #b_IDLE )
      wire#w1
      R_Coil( #P_CMD )
   END_RUNG
   RUNG wire#w1
      R_Coil( #V_CMD )
   END_RUNG
   RUNG wire#w1
      { S7_Templates := "[date_type := Date_And_Time, time_type := Time]" } T_DIFF(IN1 := #LDT_Finish, IN2 := #LDT_Start, OUT => #TimeDose)
   END_RUNG
   RUNG wire#w1
      { S7_GenerateENO := "TRUE" } Move(in := 0, out1 => #IQRB_STEP)
   END_RUNG
   RUNG wire#w1
      { S7_GenerateENO := "TRUE" } Move(in := #SP_IdleSPEED, out1 => #P_SPEED)
   END_RUNG
   RUNG wire#w1
      { S7_GenerateENO := "TRUE" } Move(in := 0.0, out1 => #r_SETTLE_T)
   END_RUNG
   RUNG wire#w1
      Contact( #ISTART_COND )
      Contact( #IOP_COND )
      Contact( #b_START )
      { S7_GenerateENO := "TRUE" } Move(in := 10, out1 => #CMD_STEP)
   END_RUNG
   // the same network as SCL:
   IF #b_IDLE THEN
       #P_CMD := FALSE;
       #V_CMD := FALSE;
       T_DIFF(IN1 := #LDT_Finish, IN2 := #LDT_Start, OUT => #TimeDose);
       #IQRB_STEP := 0;
       #P_SPEED := #SP_IdleSPEED;
       #r_SETTLE_T := 0.0;
   END_IF;
   IF #b_IDLE AND #ISTART_COND AND #IOP_COND AND #b_START THEN #CMD_STEP := 10; END_IF;
END_REGION

REGION Network 20: STEP 10: RESET COUNTER AND CALCULATE FINE AND STOP QUANTITY
   RUNG wire#powerrail
      { S7_Templates := "SrcType := Int" } EQ_Contact(in1 := #IQSTEP, in2 := 10)
      wire#w1
      { S7_GenerateENO := "TRUE" } Move(in := 10, out1 => #IQRB_STEP)
   END_RUNG
   RUNG wire#w1
      P_Trig( #PE_LDTStore )
      Move(in := #TimeDose, out1 => #LastTimeDose)
   END_RUNG
   RUNG wire#w1
      Coil( #COUNT_RESET )
   END_RUNG
   RUNG wire#w1
      { S7_GenerateENO := "TRUE" } Move(in := #IQINFL_QTY, out1 => #r_INFLIGHT)
   END_RUNG
   RUNG wire#w1
      { S7_Templates := "SrcType := Real"; S7_GenerateENO := "TRUE" } Sub(in1 := #r_STOP, in2 := #SP_FINEQTY, out => #r_FINE)
   END_RUNG
   RUNG wire#w1
      { S7_Templates := "SrcType := Real" } LE_Contact(in1 := #ACT_QTY, in2 := 0.0)
      { S7_GenerateENO := "TRUE" } Move(in := 20, out1 => #CMD_STEP)
   END_RUNG
   // the same network as SCL:
   #_w1 := #IQSTEP = 10;
   IF #_w1 THEN #IQRB_STEP := 10; END_IF;
   #_w2 := #_w1 AND NOT #PE_LDTStore;   // rising edge
   #PE_LDTStore := #_w1;
   IF #_w2 THEN #LastTimeDose := #TimeDose; END_IF;
   #COUNT_RESET := #_w1;
   IF #_w1 THEN
       #r_INFLIGHT := #IQINFL_QTY;
       #r_FINE := #r_STOP - #SP_FINEQTY;
   END_IF;
   IF #_w1 AND (#ACT_QTY <= 0.0) THEN #CMD_STEP := 20; END_IF;
END_REGION

REGION Network 21: STEP 20: OPEN VALVE
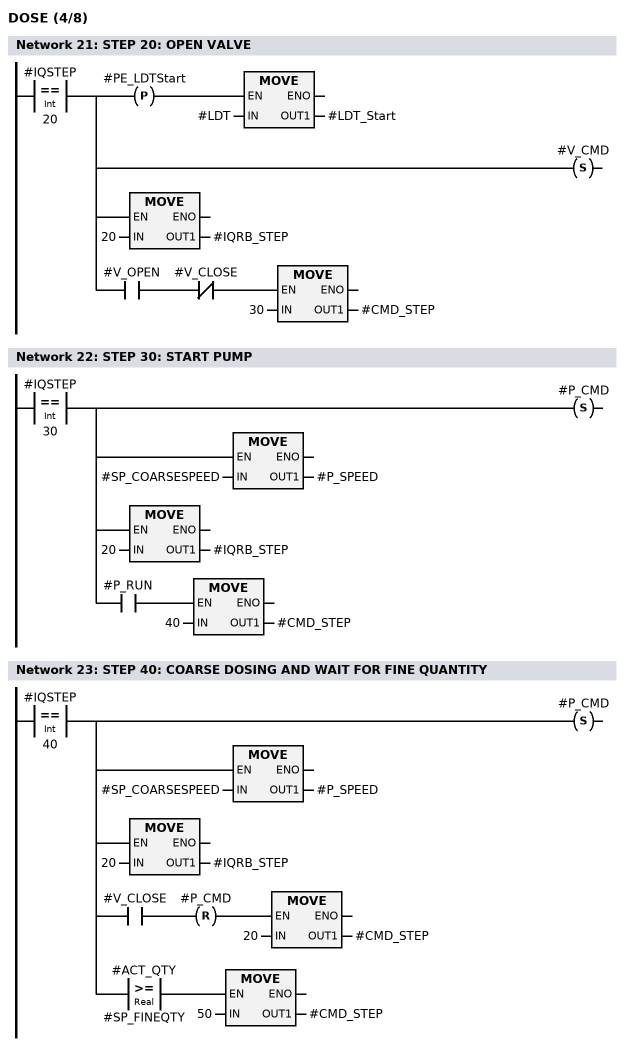
   RUNG wire#powerrail
      { S7_Templates := "SrcType := Int" } EQ_Contact(in1 := #IQSTEP, in2 := 20)
      wire#w1
      P_Trig( #PE_LDTStart )
      Move(in := #LDT, out1 => #LDT_Start)
   END_RUNG
   RUNG wire#w1
      S_Coil( #V_CMD )
   END_RUNG
   RUNG wire#w1
      { S7_GenerateENO := "TRUE" } Move(in := 20, out1 => #IQRB_STEP)
   END_RUNG
   RUNG wire#w1
      Contact( #V_OPEN )
      I_Contact( #V_CLOSE )
      { S7_GenerateENO := "TRUE" } Move(in := 30, out1 => #CMD_STEP)
   END_RUNG
   // the same network as SCL:
   #_w1 := #IQSTEP = 20;
   #_w2 := #_w1 AND NOT #PE_LDTStart;   // rising edge
   #PE_LDTStart := #_w1;
   IF #_w2 THEN #LDT_Start := #LDT; END_IF;
   IF #_w1 THEN
       #V_CMD := TRUE;
       #IQRB_STEP := 20;
   END_IF;
   IF #_w1 AND #V_OPEN AND NOT #V_CLOSE THEN #CMD_STEP := 30; END_IF;
END_REGION

REGION Network 22: STEP 30: START PUMP
   RUNG wire#powerrail
      { S7_Templates := "SrcType := Int" } EQ_Contact(in1 := #IQSTEP, in2 := 30)
      wire#w1
      S_Coil( #P_CMD )
   END_RUNG
   RUNG wire#w1
      { S7_GenerateENO := "TRUE" } Move(in := #SP_COARSESPEED, out1 => #P_SPEED)
   END_RUNG
   RUNG wire#w1
      { S7_GenerateENO := "TRUE" } Move(in := 20, out1 => #IQRB_STEP)
   END_RUNG
   RUNG wire#w1
      Contact( #P_RUN )
      { S7_GenerateENO := "TRUE" } Move(in := 40, out1 => #CMD_STEP)
   END_RUNG
   // the same network as SCL:
   #_w1 := #IQSTEP = 30;
   IF #_w1 THEN
       #P_CMD := TRUE;
       #P_SPEED := #SP_COARSESPEED;
       #IQRB_STEP := 20;
   END_IF;
   IF #_w1 AND #P_RUN THEN #CMD_STEP := 40; END_IF;
END_REGION

REGION Network 23: STEP 40: COARSE DOSING AND WAIT FOR FINE QUANTITY
   RUNG wire#powerrail
      { S7_Templates := "SrcType := Int" } EQ_Contact(in1 := #IQSTEP, in2 := 40)
      wire#w1
      S_Coil( #P_CMD )
   END_RUNG
   RUNG wire#w1
      { S7_GenerateENO := "TRUE" } Move(in := #SP_COARSESPEED, out1 => #P_SPEED)
   END_RUNG
   RUNG wire#w1
      { S7_GenerateENO := "TRUE" } Move(in := 20, out1 => #IQRB_STEP)
   END_RUNG
   RUNG wire#w1
      Contact( #V_CLOSE )
      R_Coil( #P_CMD )
      { S7_GenerateENO := "TRUE" } Move(in := 20, out1 => #CMD_STEP)
   END_RUNG
   RUNG wire#w1
      { S7_Templates := "SrcType := Real" } GE_Contact(in1 := #ACT_QTY, in2 := #SP_FINEQTY)
      { S7_GenerateENO := "TRUE" } Move(in := 50, out1 => #CMD_STEP)
   END_RUNG
   // the same network as SCL:
   #_w1 := #IQSTEP = 40;
   IF #_w1 THEN
       #P_CMD := TRUE;
       #P_SPEED := #SP_COARSESPEED;
       #IQRB_STEP := 20;
   END_IF;
   IF #_w1 AND #V_CLOSE THEN
       #P_CMD := FALSE;
       #CMD_STEP := 20;
   END_IF;
   IF #_w1 AND (#ACT_QTY >= #SP_FINEQTY) THEN #CMD_STEP := 50; END_IF;
END_REGION

REGION Network 24: STEP 50: FINE DOSING AND WAIT FOR STOP QUANTITY
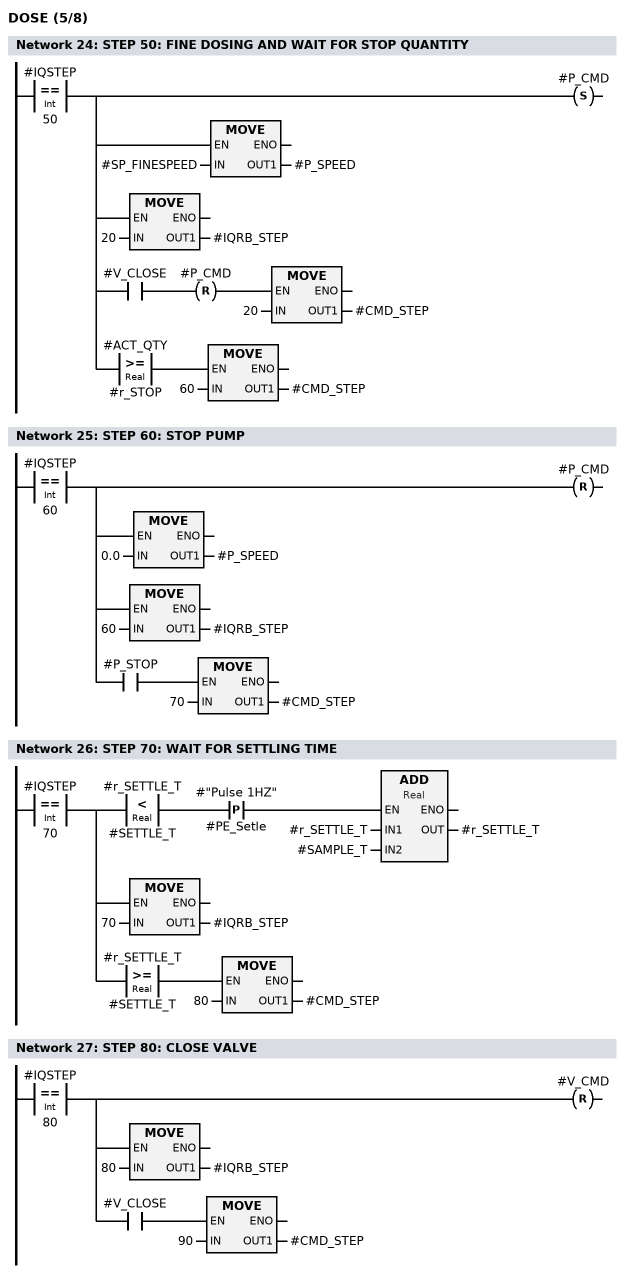
   RUNG wire#powerrail
      { S7_Templates := "SrcType := Int" } EQ_Contact(in1 := #IQSTEP, in2 := 50)
      wire#w1
      S_Coil( #P_CMD )
   END_RUNG
   RUNG wire#w1
      { S7_GenerateENO := "TRUE" } Move(in := #SP_FINESPEED, out1 => #P_SPEED)
   END_RUNG
   RUNG wire#w1
      { S7_GenerateENO := "TRUE" } Move(in := 20, out1 => #IQRB_STEP)
   END_RUNG
   RUNG wire#w1
      Contact( #V_CLOSE )
      R_Coil( #P_CMD )
      { S7_GenerateENO := "TRUE" } Move(in := 20, out1 => #CMD_STEP)
   END_RUNG
   RUNG wire#w1
      { S7_Templates := "SrcType := Real" } GE_Contact(in1 := #ACT_QTY, in2 := #r_STOP)
      { S7_GenerateENO := "TRUE" } Move(in := 60, out1 => #CMD_STEP)
   END_RUNG
   // the same network as SCL:
   #_w1 := #IQSTEP = 50;
   IF #_w1 THEN
       #P_CMD := TRUE;
       #P_SPEED := #SP_FINESPEED;
       #IQRB_STEP := 20;
   END_IF;
   IF #_w1 AND #V_CLOSE THEN
       #P_CMD := FALSE;
       #CMD_STEP := 20;
   END_IF;
   IF #_w1 AND (#ACT_QTY >= #r_STOP) THEN #CMD_STEP := 60; END_IF;
END_REGION

REGION Network 25: STEP 60: STOP PUMP
   RUNG wire#powerrail
      { S7_Templates := "SrcType := Int" } EQ_Contact(in1 := #IQSTEP, in2 := 60)
      wire#w1
      R_Coil( #P_CMD )
   END_RUNG
   RUNG wire#w1
      { S7_GenerateENO := "TRUE" } Move(in := 0.0, out1 => #P_SPEED)
   END_RUNG
   RUNG wire#w1
      { S7_GenerateENO := "TRUE" } Move(in := 60, out1 => #IQRB_STEP)
   END_RUNG
   RUNG wire#w1
      Contact( #P_STOP )
      { S7_GenerateENO := "TRUE" } Move(in := 70, out1 => #CMD_STEP)
   END_RUNG
   // the same network as SCL:
   #_w1 := #IQSTEP = 60;
   IF #_w1 THEN
       #P_CMD := FALSE;
       #P_SPEED := 0.0;
       #IQRB_STEP := 60;
   END_IF;
   IF #_w1 AND #P_STOP THEN #CMD_STEP := 70; END_IF;
END_REGION

REGION Network 26: STEP 70: WAIT FOR SETTLING TIME
   RUNG wire#powerrail
      { S7_Templates := "SrcType := Int" } EQ_Contact(in1 := #IQSTEP, in2 := 70)
      wire#w1
      { S7_Templates := "SrcType := Real" } LT_Contact(in1 := #r_SETTLE_T, in2 := #SETTLE_T)
      P_Contact(operand := #"Pulse 1HZ", bit := #PE_Setle)
      { S7_Templates := "SrcType := Real"; S7_GenerateENO := "TRUE" } Add(in1 := #r_SETTLE_T, in2 := #SAMPLE_T, out => #r_SETTLE_T)
   END_RUNG
   RUNG wire#w1
      { S7_GenerateENO := "TRUE" } Move(in := 70, out1 => #IQRB_STEP)
   END_RUNG
   RUNG wire#w1
      { S7_Templates := "SrcType := Real" } GE_Contact(in1 := #r_SETTLE_T, in2 := #SETTLE_T)
      { S7_GenerateENO := "TRUE" } Move(in := 80, out1 => #CMD_STEP)
   END_RUNG
   // the same network as SCL:
   #_w1 := #IQSTEP = 70;
   #_w2 := #_w1 AND (#r_SETTLE_T < #SETTLE_T) AND #"Pulse 1HZ" AND NOT #PE_Setle;   // rising edge of #"Pulse 1HZ"
   #PE_Setle := #"Pulse 1HZ";
   IF #_w2 THEN #r_SETTLE_T := #r_SETTLE_T + #SAMPLE_T; END_IF;
   IF #_w1 THEN #IQRB_STEP := 70; END_IF;
   IF #_w1 AND (#r_SETTLE_T >= #SETTLE_T) THEN #CMD_STEP := 80; END_IF;
END_REGION

REGION Network 27: STEP 80: CLOSE VALVE
   RUNG wire#powerrail
      { S7_Templates := "SrcType := Int" } EQ_Contact(in1 := #IQSTEP, in2 := 80)
      wire#w1
      R_Coil( #V_CMD )
   END_RUNG
   RUNG wire#w1
      { S7_GenerateENO := "TRUE" } Move(in := 80, out1 => #IQRB_STEP)
   END_RUNG
   RUNG wire#w1
      Contact( #V_CLOSE )
      { S7_GenerateENO := "TRUE" } Move(in := 90, out1 => #CMD_STEP)
   END_RUNG
   // the same network as SCL:
   #_w1 := #IQSTEP = 80;
   IF #_w1 THEN
       #V_CMD := FALSE;
       #IQRB_STEP := 80;
   END_IF;
   IF #_w1 AND #V_CLOSE THEN #CMD_STEP := 90; END_IF;
END_REGION

REGION Network 28: STEP 90: CALCULATE INFLIGHT QTY
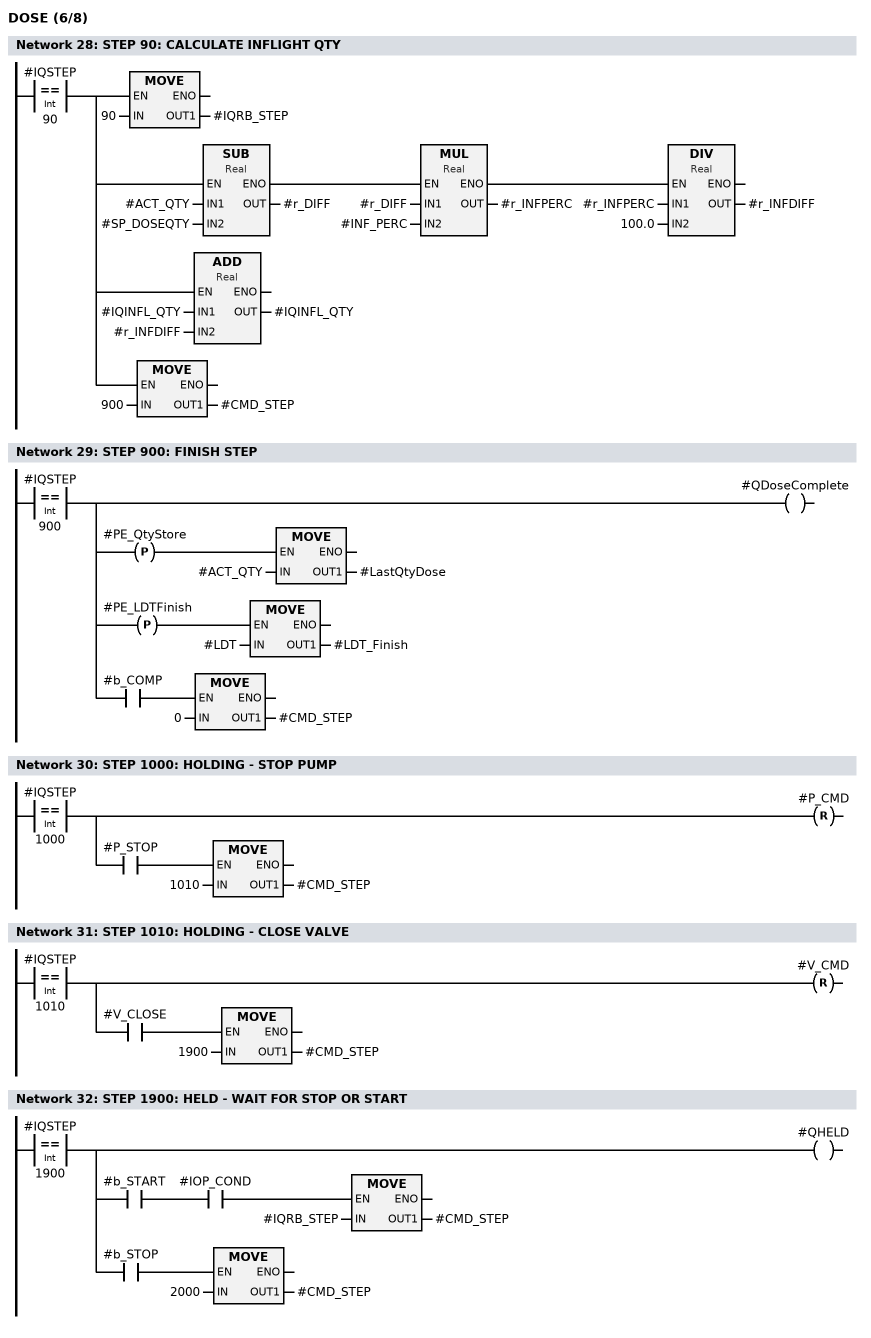
   RUNG wire#powerrail
      { S7_Templates := "SrcType := Int" } EQ_Contact(in1 := #IQSTEP, in2 := 90)
      wire#w1
      { S7_GenerateENO := "TRUE" } Move(in := 90, out1 => #IQRB_STEP)
   END_RUNG
   RUNG wire#w1
      { S7_Templates := "SrcType := Real"; S7_GenerateENO := "TRUE" } Sub(in1 := #ACT_QTY, in2 := #SP_DOSEQTY, out => #r_DIFF)
      { S7_Templates := "SrcType := Real"; S7_GenerateENO := "TRUE" } Mul(in1 := #r_DIFF, in2 := #INF_PERC, out => #r_INFPERC)
      { S7_Templates := "SrcType := Real"; S7_GenerateENO := "TRUE" } Div(in1 := #r_INFPERC, in2 := 100.0, out => #r_INFDIFF)
   END_RUNG
   RUNG wire#w1
      { S7_Templates := "SrcType := Real"; S7_GenerateENO := "TRUE" } Add(in1 := #IQINFL_QTY, in2 := #r_INFDIFF, out => #IQINFL_QTY)
   END_RUNG
   RUNG wire#w1
      { S7_GenerateENO := "TRUE" } Move(in := 900, out1 => #CMD_STEP)
   END_RUNG
   // the same network as SCL:
   // ENO of a box is taken as its EN; it also drops when the box reports an error
   IF #IQSTEP = 90 THEN
       #IQRB_STEP := 90;
       #r_DIFF := #ACT_QTY - #SP_DOSEQTY;
       #r_INFPERC := #r_DIFF * #INF_PERC;
       #r_INFDIFF := #r_INFPERC / 100.0;
       #IQINFL_QTY := #IQINFL_QTY + #r_INFDIFF;
       #CMD_STEP := 900;
   END_IF;
END_REGION

REGION Network 29: STEP 900: FINISH STEP
   RUNG wire#powerrail
      { S7_Templates := "SrcType := Int" } EQ_Contact(in1 := #IQSTEP, in2 := 900)
      wire#w1
      Coil( #QDoseComplete )
   END_RUNG
   RUNG wire#w1
      P_Trig( #PE_QtyStore )
      Move(in := #ACT_QTY, out1 => #LastQtyDose)
   END_RUNG
   RUNG wire#w1
      P_Trig( #PE_LDTFinish )
      Move(in := #LDT, out1 => #LDT_Finish)
   END_RUNG
   RUNG wire#w1
      Contact( #b_COMP )
      { S7_GenerateENO := "TRUE" } Move(in := 0, out1 => #CMD_STEP)
   END_RUNG
   // the same network as SCL:
   #QDoseComplete := #IQSTEP = 900;
   #_w1 := #QDoseComplete AND NOT #PE_QtyStore;   // rising edge
   #PE_QtyStore := #QDoseComplete;
   IF #_w1 THEN #LastQtyDose := #ACT_QTY; END_IF;
   #_w2 := #QDoseComplete AND NOT #PE_LDTFinish;   // rising edge
   #PE_LDTFinish := #QDoseComplete;
   IF #_w2 THEN #LDT_Finish := #LDT; END_IF;
   IF #QDoseComplete AND #b_COMP THEN #CMD_STEP := 0; END_IF;
END_REGION

REGION Network 30: STEP 1000: HOLDING - STOP PUMP
   RUNG wire#powerrail
      { S7_Templates := "SrcType := Int" } EQ_Contact(in1 := #IQSTEP, in2 := 1000)
      wire#w1
      R_Coil( #P_CMD )
   END_RUNG
   RUNG wire#w1
      Contact( #P_STOP )
      { S7_GenerateENO := "TRUE" } Move(in := 1010, out1 => #CMD_STEP)
   END_RUNG
   // the same network as SCL:
   #_w1 := #IQSTEP = 1000;
   IF #_w1 THEN #P_CMD := FALSE; END_IF;
   IF #_w1 AND #P_STOP THEN #CMD_STEP := 1010; END_IF;
END_REGION

REGION Network 31: STEP 1010: HOLDING - CLOSE VALVE
   RUNG wire#powerrail
      { S7_Templates := "SrcType := Int" } EQ_Contact(in1 := #IQSTEP, in2 := 1010)
      wire#w1
      R_Coil( #V_CMD )
   END_RUNG
   RUNG wire#w1
      Contact( #V_CLOSE )
      { S7_GenerateENO := "TRUE" } Move(in := 1900, out1 => #CMD_STEP)
   END_RUNG
   // the same network as SCL:
   #_w1 := #IQSTEP = 1010;
   IF #_w1 THEN #V_CMD := FALSE; END_IF;
   IF #_w1 AND #V_CLOSE THEN #CMD_STEP := 1900; END_IF;
END_REGION

REGION Network 32: STEP 1900: HELD - WAIT FOR STOP OR START
   RUNG wire#powerrail
      { S7_Templates := "SrcType := Int" } EQ_Contact(in1 := #IQSTEP, in2 := 1900)
      wire#w1
      Coil( #QHELD )
   END_RUNG
   RUNG wire#w1
      Contact( #b_START )
      Contact( #IOP_COND )
      { S7_GenerateENO := "TRUE" } Move(in := #IQRB_STEP, out1 => #CMD_STEP)
   END_RUNG
   RUNG wire#w1
      Contact( #b_STOP )
      { S7_GenerateENO := "TRUE" } Move(in := 2000, out1 => #CMD_STEP)
   END_RUNG
   // the same network as SCL:
   #QHELD := #IQSTEP = 1900;
   IF #QHELD AND #b_START AND #IOP_COND THEN #CMD_STEP := #IQRB_STEP; END_IF;
   IF #QHELD AND #b_STOP THEN #CMD_STEP := 2000; END_IF;
END_REGION

REGION Network 33: STEP 2000: STOPPING - STOP PUMP
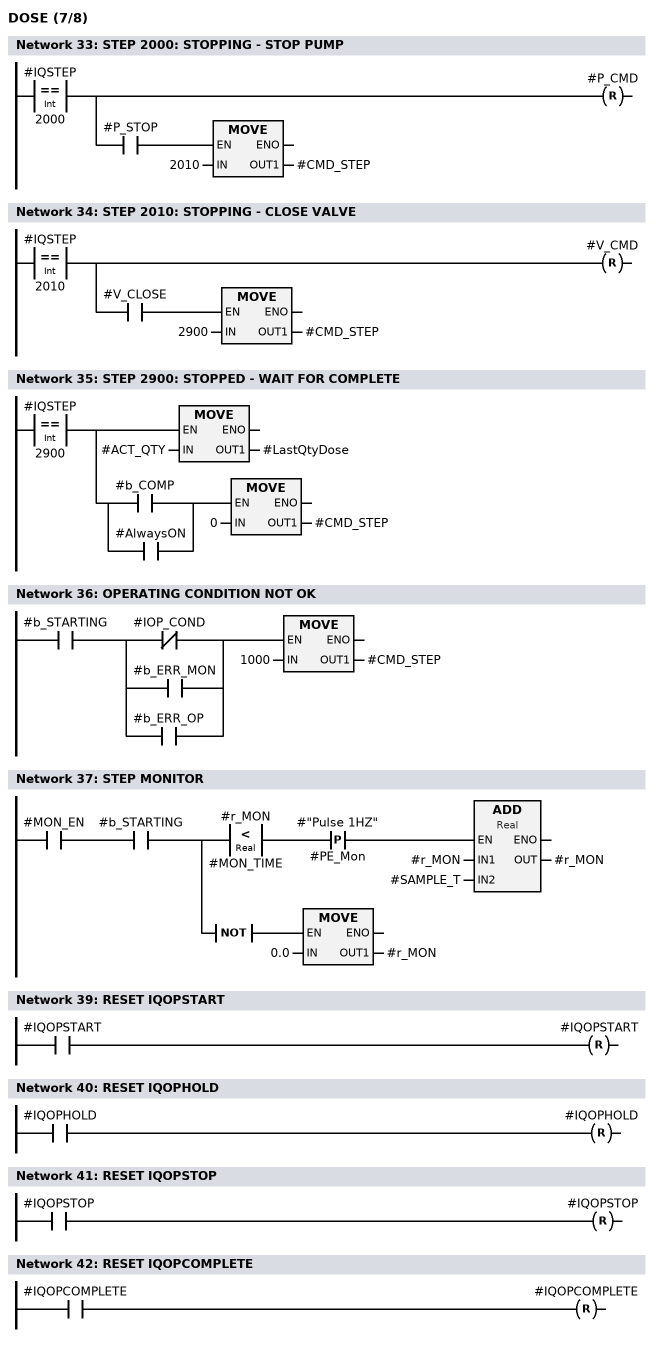
   RUNG wire#powerrail
      { S7_Templates := "SrcType := Int" } EQ_Contact(in1 := #IQSTEP, in2 := 2000)
      wire#w1
      R_Coil( #P_CMD )
   END_RUNG
   RUNG wire#w1
      Contact( #P_STOP )
      { S7_GenerateENO := "TRUE" } Move(in := 2010, out1 => #CMD_STEP)
   END_RUNG
   // the same network as SCL:
   #_w1 := #IQSTEP = 2000;
   IF #_w1 THEN #P_CMD := FALSE; END_IF;
   IF #_w1 AND #P_STOP THEN #CMD_STEP := 2010; END_IF;
END_REGION

REGION Network 34: STEP 2010: STOPPING - CLOSE VALVE
   RUNG wire#powerrail
      { S7_Templates := "SrcType := Int" } EQ_Contact(in1 := #IQSTEP, in2 := 2010)
      wire#w1
      R_Coil( #V_CMD )
   END_RUNG
   RUNG wire#w1
      Contact( #V_CLOSE )
      { S7_GenerateENO := "TRUE" } Move(in := 2900, out1 => #CMD_STEP)
   END_RUNG
   // the same network as SCL:
   #_w1 := #IQSTEP = 2010;
   IF #_w1 THEN #V_CMD := FALSE; END_IF;
   IF #_w1 AND #V_CLOSE THEN #CMD_STEP := 2900; END_IF;
END_REGION

REGION Network 35: STEP 2900: STOPPED - WAIT FOR COMPLETE
   RUNG wire#powerrail
      { S7_Templates := "SrcType := Int" } EQ_Contact(in1 := #IQSTEP, in2 := 2900)
      wire#w1
      Move(in := #ACT_QTY, out1 => #LastQtyDose)
   END_RUNG
   RUNG wire#w1
      Contact( #b_COMP )
      wire#w2
      { S7_GenerateENO := "TRUE" } Move(in := 0, out1 => #CMD_STEP)
   END_RUNG
   RUNG wire#w1
      Contact( #AlwaysON )
   END_RUNG wire#w2
   // the same network as SCL:
   #_w1 := #IQSTEP = 2900;
   IF #_w1 THEN #LastQtyDose := #ACT_QTY; END_IF;
   IF #_w1 AND (#b_COMP OR #AlwaysON) THEN #CMD_STEP := 0; END_IF;
END_REGION

REGION Network 36: OPERATING CONDITION NOT OK
   RUNG wire#powerrail
      Contact( #b_STARTING )
      wire#w1
      I_Contact( #IOP_COND )
      wire#w2
      { S7_GenerateENO := "TRUE" } Move(in := 1000, out1 => #CMD_STEP)
   END_RUNG
   RUNG wire#w1
      Contact( #b_ERR_MON )
   END_RUNG wire#w2
   RUNG wire#w1
      Contact( #b_ERR_OP )
   END_RUNG wire#w2
   // the same network as SCL:
   IF #b_STARTING AND (NOT #IOP_COND OR #b_ERR_MON OR #b_ERR_OP) THEN #CMD_STEP := 1000; END_IF;
END_REGION

REGION Network 37: STEP MONITOR
   RUNG wire#powerrail
      Contact( #MON_EN )
      Contact( #b_STARTING )
      wire#w1
      { S7_Templates := "SrcType := Real" } LT_Contact(in1 := #r_MON, in2 := #MON_TIME)
      P_Contact(operand := #"Pulse 1HZ", bit := #PE_Mon)
      { S7_Templates := "SrcType := Real"; S7_GenerateENO := "TRUE" } Add(in1 := #r_MON, in2 := #SAMPLE_T, out => #r_MON)
   END_RUNG
   RUNG wire#w1
      Not()
      { S7_GenerateENO := "TRUE" } Move(in := 0.0, out1 => #r_MON)
   END_RUNG
   // the same network as SCL:
   #_w1 := #MON_EN AND #b_STARTING;
   #_w2 := #_w1 AND (#r_MON < #MON_TIME) AND #"Pulse 1HZ" AND NOT #PE_Mon;   // rising edge of #"Pulse 1HZ"
   #PE_Mon := #"Pulse 1HZ";
   IF #_w2 THEN #r_MON := #r_MON + #SAMPLE_T; END_IF;
   IF NOT #_w1 THEN #r_MON := 0.0; END_IF;
END_REGION

REGION Network 38: RESET IQRESET
END_REGION

REGION Network 39: RESET IQOPSTART
   RUNG wire#powerrail
      Contact( #IQOPSTART )
      R_Coil( #IQOPSTART )
   END_RUNG
   // the same network as SCL:
   IF #IQOPSTART THEN #IQOPSTART := FALSE; END_IF;
END_REGION

REGION Network 40: RESET IQOPHOLD
   RUNG wire#powerrail
      Contact( #IQOPHOLD )
      R_Coil( #IQOPHOLD )
   END_RUNG
   // the same network as SCL:
   IF #IQOPHOLD THEN #IQOPHOLD := FALSE; END_IF;
END_REGION

REGION Network 41: RESET IQOPSTOP
   RUNG wire#powerrail
      Contact( #IQOPSTOP )
      R_Coil( #IQOPSTOP )
   END_RUNG
   // the same network as SCL:
   IF #IQOPSTOP THEN #IQOPSTOP := FALSE; END_IF;
END_REGION

REGION Network 42: RESET IQOPCOMPLETE
   RUNG wire#powerrail
      Contact( #IQOPCOMPLETE )
      R_Coil( #IQOPCOMPLETE )
   END_RUNG
   // the same network as SCL:
   IF #IQOPCOMPLETE THEN #IQOPCOMPLETE := FALSE; END_IF;
END_REGION

REGION Network 43: DOSED QUANTITY
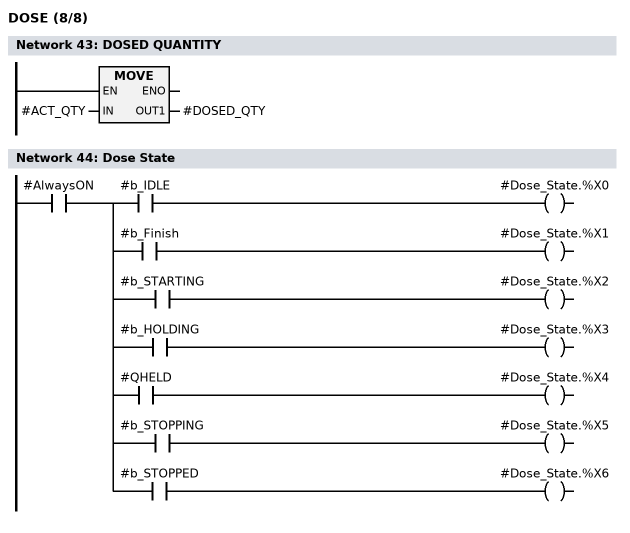
   RUNG wire#powerrail
      { S7_GenerateENO := "TRUE" } Move(in := #ACT_QTY, out1 => #DOSED_QTY)
   END_RUNG
   // the same network as SCL:
   #DOSED_QTY := #ACT_QTY;
END_REGION

REGION Network 44: Dose State
   RUNG wire#powerrail
      Contact( #AlwaysON )
      wire#w1
      Contact( #b_IDLE )
      Coil( #Dose_State.%X0 )
   END_RUNG
   RUNG wire#w1
      Contact( #b_Finish )
      Coil( #Dose_State.%X1 )
   END_RUNG
   RUNG wire#w1
      Contact( #b_STARTING )
      Coil( #Dose_State.%X2 )
   END_RUNG
   RUNG wire#w1
      Contact( #b_HOLDING )
      Coil( #Dose_State.%X3 )
   END_RUNG
   RUNG wire#w1
      Contact( #QHELD )
      Coil( #Dose_State.%X4 )
   END_RUNG
   RUNG wire#w1
      Contact( #b_STOPPING )
      Coil( #Dose_State.%X5 )
   END_RUNG
   RUNG wire#w1
      Contact( #b_STOPPED )
      Coil( #Dose_State.%X6 )
   END_RUNG
   // the same network as SCL:
   #Dose_State.%X0 := #AlwaysON AND #b_IDLE;
   #Dose_State.%X1 := #AlwaysON AND #b_Finish;
   #Dose_State.%X2 := #AlwaysON AND #b_STARTING;
   #Dose_State.%X3 := #AlwaysON AND #b_HOLDING;
   #Dose_State.%X4 := #AlwaysON AND #QHELD;
   #Dose_State.%X5 := #AlwaysON AND #b_STOPPING;
   #Dose_State.%X6 := #AlwaysON AND #b_STOPPED;
END_REGION
END_FUNCTION_BLOCK

FUNCTION_BLOCK "BFT_ChiliFresh"   // FB364, LAD
{ S7_Optimized_Access := 'TRUE' }
VERSION : 0.1
// stored: AutoNumber false, IsIECCheckEnabled false, IsRetainMemResEnabled false, MemoryReserve 100, SetENOAutomatically false, UDAEnableTagReadback false
   VAR_INPUT
      IN_FBAV_Inload : Bool;
      IN_FBAV_Outlet : Bool;
      IN_FBAV_Transfer : Bool;
      IN_FBAV_CIP_Tank : Bool;
      IN_FBAV_CIP_Line : Bool;
      IN_FBP_Inload : Bool;
      IN_FBP_Inload_SP : Real;
      IN_FBP_Transfer : Bool;
      IN_FBP_Transfer_SP : Real;
      IN_FBP_CIP : Bool;
      IN_FBP_CIP_Sp : Real;
      IN_LT01 : Real;
      "LCS Start" : Bool;
      "LCS Stop" : Bool;
      "LCS EMS" : Bool;
      IN_Dose_Run : Bool;
      IN_Dose_Held : Bool;
      IN_Dose_Complete : Bool;
      IN_Dose_Header_1 : Bool;
      IN_Dose_Header_2 : Bool;
      IN_Dose_Valve_Cmd : Bool;
      IN_Dose_Pump_Cmd : Bool;
      IN_Dose_Pump_Sp : Real;
      IN_Dose_LineOK : Bool;
      "Inload Busy" : Bool;
      IN_Prod_Ready : Bool;
      IN_Prod_LineOpen : Bool;
      IN_Prod_SupplyOn : Bool;
      IN_Prod_Transfer_Comp : Bool;
      "CIP Pulse" : Bool;
      "CIP Supply ON" : Bool;
      "CIP Req OK" : Bool;
      "CIP Complete" : Bool;
      "CIP Busy" : Bool;
   END_VAR
   VAR_OUTPUT
      Out_AV_Inload : Bool;
      Out_AV_Outlet : Bool;
      Out_AV_Transfer : Bool;
      Out_AV_CIP_Tank : Bool;
      Out_AV_CIP_Line : Bool;
      Out_P_Inload : Bool;
      Out_P_Inload_Sp : Real;
      Out_P_Transfer : Bool;
      Out_P_Transfer_Sp : Real;
      Out_P_CIP : Bool;
      Out_P_CIP_Sp : Real;
      Out_Prod_Req : Bool;
      Out_Prod_LineOpen : Bool;
      Out_CIP_Req : Bool;
      Out_CIP_LineOpen : Bool;
   END_VAR
   VAR
      Cmd : Struct
         Inload : Bool;
         Ready_for_Tranfer : Bool;
         CIP_Tank : Bool;
         CIP_Line : Bool;
      END_STRUCT;
   END_VAR
   VAR RETAIN
      Param : Struct
         SP_Level_LL : Real := 10.0;
         SP_Level_ML : Real := 80.0;
         SP_Level_HL : Real := 100.0;
         SupplyPump_SP_Speed : Real := 80.0;
         L_Hi_Lim : Real := 100.0;
         L_Lo_Lim : Real := 0.0;
         L_Hys : Real := 2.0;
         FlushingTime : DInt := 10000;
         CIP_Trf_SP_Speed : Real := 80.0;
         CIP_Ret_ON_SP : Real := 5.0;
         CIP_Ret_OFF_SP : Real;
      END_STRUCT;
   END_VAR
   VAR
      State : Struct   // Tank in loading state
         Tank_LL : Bool;
         Tank_ML : Bool;
         Tank_HL : Bool;
         Tank_inCIP : Bool;
         Tank_CIP_Enable : Bool;
         Line_inCIP : Bool;
         Line_CIP_Enable : Bool;
         CIP_Return_On : Bool;
         Inloading : Bool;
         Inload_Enable : Bool;
         Ready_For_Transfer : Bool;
         Ready_For_Transfer_Ena : Bool;
         Tank_Available : Bool;
         Transfer_On_Prog : Bool;
      END_STRUCT;
      alwaysON : Bool;
      L_Hys_Abs : Real;
      Hys_Level_HL : Real;
      Hys_Level_ML : Real;
      Hys_Level_LL : Real;
      r : Struct
         PosE1 : Bool;
         PosE2 : Bool;
         PosE3 : Bool;
         PosE4 : Bool;
         PosE5 : Bool;
         PosE6 : Bool;
         PosE7 : Bool;
         PosE8 : Bool;
         PosE9 : Bool;
         PosE10 : Bool;
         PosE11 : Bool;
         PosE12 : Bool;
         PosE13 : Bool;
         PosE14 : Bool;
         PosE15 : Bool;
         PosE16 : Bool;
         PosE17 : Bool;
         PosE18 : Bool;
         PosE19 : Bool;
         PosE20 : Bool;
         PosE21 : Bool;
         PosE22 : Bool;
         PosE23 : Bool;
         PosE24 : Bool;
         PosE25 : Bool;
         PosE26 : Bool;
         PosE27 : Bool;
         PosE28 : Bool;
         PosE29 : Bool;
         PosE30 : Bool;
         PosE31 : Bool;
         PosE32 : Bool;
      END_STRUCT;
      Actuator : Struct
         AV_Inload : Bool;
         AV_Outlet : Bool;
         AV_Transfer : Bool;
         AV_CIP_Tank : Bool;
         AV_CIP_Line : Bool;
         P_Transfer : Bool;
         P_Inload : Bool;
         P_CIP : Bool;
      END_STRUCT;
      FlushingTim : TON_TIME;
      SPumpTim { S7_SetPoint := 'True'} : TON_TIME;
      AVinloadTim { S7_SetPoint := 'True'} : TON_TIME;
      Pump_TF_On_Time { S7_SetPoint := 'True'} : TON_TIME;
   END_VAR
   VAR_TEMP   // added for the SCL form of the ladder/FBD networks
      _w1 : Bool;
      _w2 : Bool;
   END_VAR
BEGIN

REGION Network 1: Always_ON
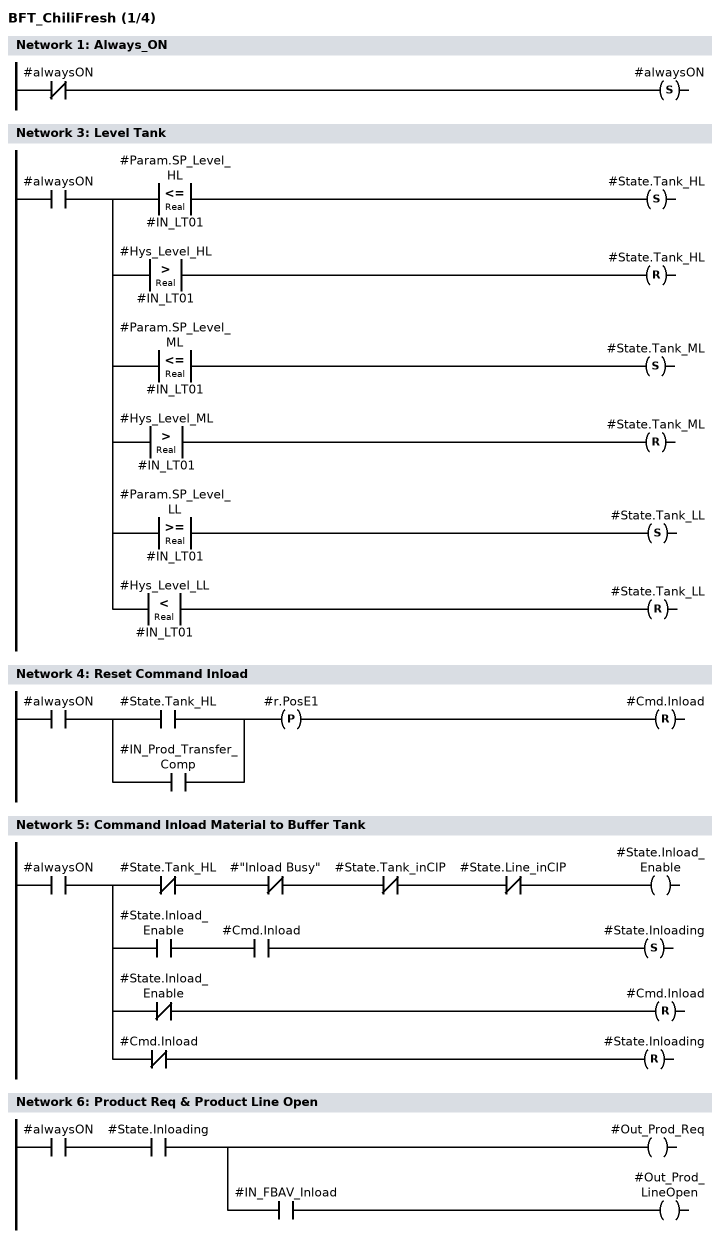
   RUNG wire#powerrail
      I_Contact( #alwaysON )
      S_Coil( #alwaysON )
   END_RUNG
   // the same network as SCL:
   IF NOT #alwaysON THEN #alwaysON := TRUE; END_IF;
END_REGION

NETWORK
TITLE = Hys Calculation
//Level Hys Absolute
      L     #Param.L_Hi_Lim;
      L     #Param.L_Lo_Lim;
      -R;
      L     100.0;
      /R;
      L     #Param.L_Hys;
      *R;
      T     #L_Hys_Abs;
//Tank High Level
      L     #Param.SP_Level_HL;
      L     #L_Hys_Abs;
      -R;
      T     #Hys_Level_HL;
//Tank Mid Level
      L     #Param.SP_Level_ML;
      L     #L_Hys_Abs;
      -R;
      T     #Hys_Level_ML;
//Tank Low Level
      L     #Param.SP_Level_LL;
      L     #L_Hys_Abs;
      +R;
      T     #Hys_Level_LL;


REGION Network 3: Level Tank
   RUNG wire#powerrail
      Contact( #alwaysON )
      wire#w1
      { S7_Templates := "SrcType := Real" } LE_Contact(in1 := #Param.SP_Level_HL, in2 := #IN_LT01)
      S_Coil( #State.Tank_HL )
   END_RUNG
   RUNG wire#w1
      { S7_Templates := "SrcType := Real" } GT_Contact(in1 := #Hys_Level_HL, in2 := #IN_LT01)
      R_Coil( #State.Tank_HL )
   END_RUNG
   RUNG wire#w1
      { S7_Templates := "SrcType := Real" } LE_Contact(in1 := #Param.SP_Level_ML, in2 := #IN_LT01)
      S_Coil( #State.Tank_ML )
   END_RUNG
   RUNG wire#w1
      { S7_Templates := "SrcType := Real" } GT_Contact(in1 := #Hys_Level_ML, in2 := #IN_LT01)
      R_Coil( #State.Tank_ML )
   END_RUNG
   RUNG wire#w1
      { S7_Templates := "SrcType := Real" } GE_Contact(in1 := #Param.SP_Level_LL, in2 := #IN_LT01)
      S_Coil( #State.Tank_LL )
   END_RUNG
   RUNG wire#w1
      { S7_Templates := "SrcType := Real" } LT_Contact(in1 := #Hys_Level_LL, in2 := #IN_LT01)
      R_Coil( #State.Tank_LL )
   END_RUNG
   // the same network as SCL:
   IF #alwaysON AND (#Param.SP_Level_HL <= #IN_LT01) THEN #State.Tank_HL := TRUE; END_IF;
   IF #alwaysON AND (#Hys_Level_HL > #IN_LT01) THEN #State.Tank_HL := FALSE; END_IF;
   IF #alwaysON AND (#Param.SP_Level_ML <= #IN_LT01) THEN #State.Tank_ML := TRUE; END_IF;
   IF #alwaysON AND (#Hys_Level_ML > #IN_LT01) THEN #State.Tank_ML := FALSE; END_IF;
   IF #alwaysON AND (#Param.SP_Level_LL >= #IN_LT01) THEN #State.Tank_LL := TRUE; END_IF;
   IF #alwaysON AND (#Hys_Level_LL < #IN_LT01) THEN #State.Tank_LL := FALSE; END_IF;
END_REGION

REGION Network 4: Reset Command Inload
   RUNG wire#powerrail
      Contact( #alwaysON )
      wire#w1
      Contact( #State.Tank_HL )
      wire#w2
      P_Trig( #r.PosE1 )
      R_Coil( #Cmd.Inload )
   END_RUNG
   RUNG wire#w1
      Contact( #IN_Prod_Transfer_Comp )
   END_RUNG wire#w2
   // the same network as SCL:
   #_w1 := #alwaysON AND (#State.Tank_HL OR #IN_Prod_Transfer_Comp);
   #_w2 := #_w1 AND NOT #r.PosE1;   // rising edge
   #r.PosE1 := #_w1;
   IF #_w2 THEN #Cmd.Inload := FALSE; END_IF;
END_REGION

REGION Network 5: Command Inload Material to Buffer Tank
   RUNG wire#powerrail
      Contact( #alwaysON )
      wire#w1
      I_Contact( #State.Tank_HL )
      I_Contact( #"Inload Busy" )
      I_Contact( #State.Tank_inCIP )
      I_Contact( #State.Line_inCIP )
      Coil( #State.Inload_Enable )
   END_RUNG
   RUNG wire#w1
      Contact( #State.Inload_Enable )
      Contact( #Cmd.Inload )
      S_Coil( #State.Inloading )
   END_RUNG
   RUNG wire#w1
      I_Contact( #State.Inload_Enable )
      R_Coil( #Cmd.Inload )
   END_RUNG
   RUNG wire#w1
      I_Contact( #Cmd.Inload )
      R_Coil( #State.Inloading )
   END_RUNG
   // the same network as SCL:
   #State.Inload_Enable := #alwaysON AND NOT #State.Tank_HL AND NOT #"Inload Busy" AND NOT #State.Tank_inCIP AND NOT #State.Line_inCIP;
   IF #alwaysON AND #State.Inload_Enable AND #Cmd.Inload THEN #State.Inloading := TRUE; END_IF;
   IF #alwaysON AND NOT #State.Inload_Enable THEN #Cmd.Inload := FALSE; END_IF;
   IF #alwaysON AND NOT #Cmd.Inload THEN #State.Inloading := FALSE; END_IF;
END_REGION

REGION Network 6: Product Req & Product Line Open
   RUNG wire#powerrail
      Contact( #alwaysON )
      Contact( #State.Inloading )
      wire#w1
      Coil( #Out_Prod_Req )
   END_RUNG
   RUNG wire#w1
      Contact( #IN_FBAV_Inload )
      Coil( #Out_Prod_LineOpen )
   END_RUNG
   // the same network as SCL:
   #Out_Prod_Req := #alwaysON AND #State.Inloading;
   #Out_Prod_LineOpen := #Out_Prod_Req AND #IN_FBAV_Inload;
END_REGION

REGION Network 8: Tank Ready for Transfer to Blending
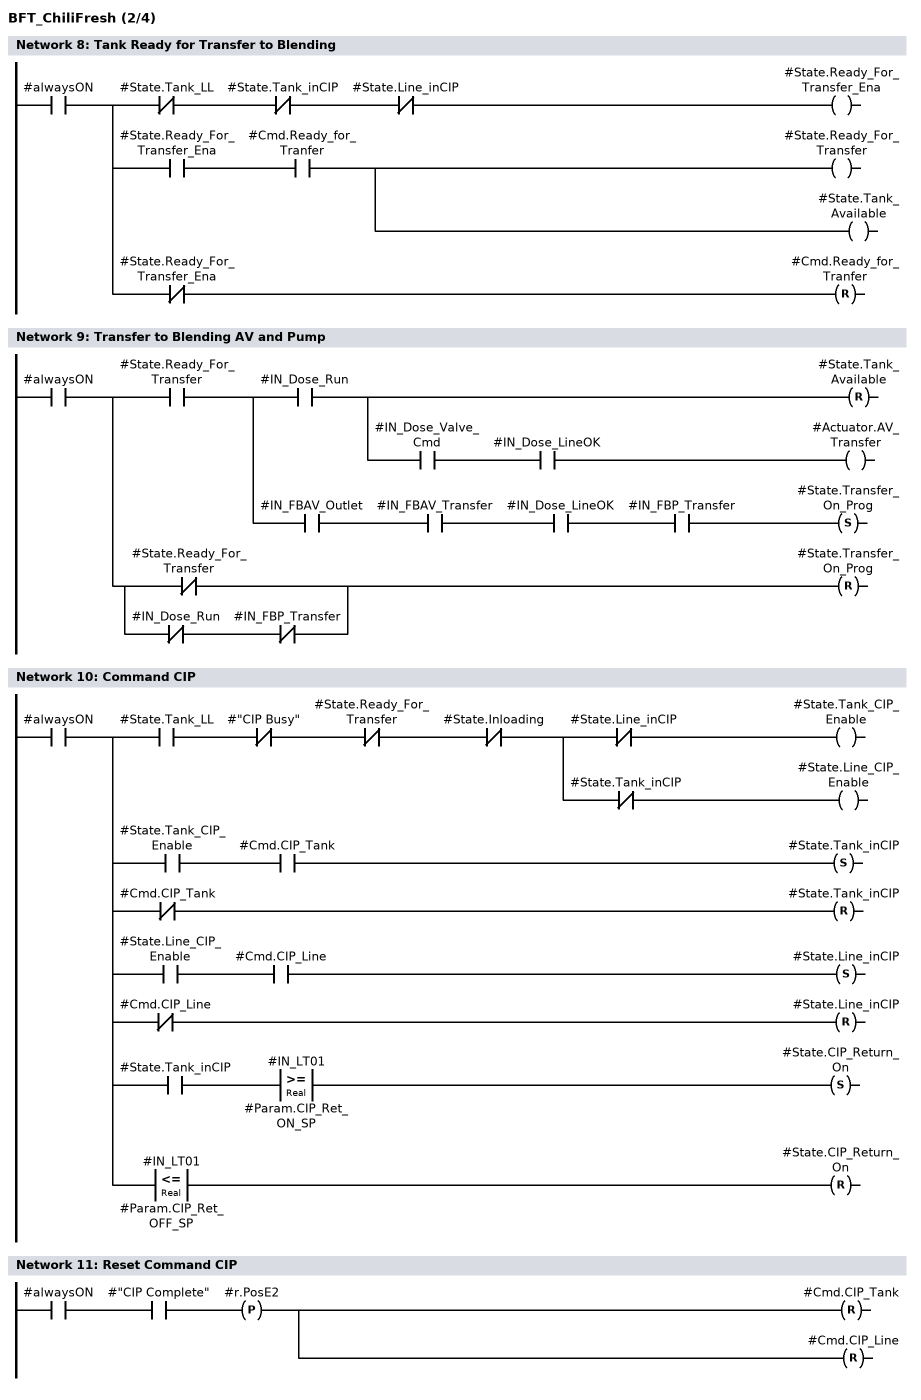
   RUNG wire#powerrail
      Contact( #alwaysON )
      wire#w1
      I_Contact( #State.Tank_LL )
      I_Contact( #State.Tank_inCIP )
      I_Contact( #State.Line_inCIP )
      Coil( #State.Ready_For_Transfer_Ena )
   END_RUNG
   RUNG wire#w1
      Contact( #State.Ready_For_Transfer_Ena )
      Contact( #Cmd.Ready_for_Tranfer )
      wire#w2
      Coil( #State.Ready_For_Transfer )
   END_RUNG
   RUNG wire#w2
      Coil( #State.Tank_Available )
   END_RUNG
   RUNG wire#w1
      I_Contact( #State.Ready_For_Transfer_Ena )
      R_Coil( #Cmd.Ready_for_Tranfer )
   END_RUNG
   // the same network as SCL:
   #State.Ready_For_Transfer_Ena := #alwaysON AND NOT #State.Tank_LL AND NOT #State.Tank_inCIP AND NOT #State.Line_inCIP;
   #State.Ready_For_Transfer := #alwaysON AND #State.Ready_For_Transfer_Ena AND #Cmd.Ready_for_Tranfer;
   #State.Tank_Available := #State.Ready_For_Transfer;
   IF #alwaysON AND NOT #State.Ready_For_Transfer_Ena THEN #Cmd.Ready_for_Tranfer := FALSE; END_IF;
END_REGION

REGION Network 9: Transfer to Blending AV and Pump
   RUNG wire#powerrail
      Contact( #alwaysON )
      wire#w1
      Contact( #State.Ready_For_Transfer )
      wire#w2
      Contact( #IN_Dose_Run )
      wire#w3
      R_Coil( #State.Tank_Available )
   END_RUNG
   RUNG wire#w3
      Contact( #IN_Dose_Valve_Cmd )
      Contact( #IN_Dose_LineOK )
      Coil( #Actuator.AV_Transfer )
   END_RUNG
   RUNG wire#w2
      Contact( #IN_FBAV_Outlet )
      Contact( #IN_FBAV_Transfer )
      Contact( #IN_Dose_LineOK )
      Contact( #IN_FBP_Transfer )
      S_Coil( #State.Transfer_On_Prog )
   END_RUNG
   RUNG wire#w1
      I_Contact( #State.Ready_For_Transfer )
      wire#w4
      R_Coil( #State.Transfer_On_Prog )
   END_RUNG
   RUNG wire#w1
      I_Contact( #IN_Dose_Run )
      I_Contact( #IN_FBP_Transfer )
   END_RUNG wire#w4
   // the same network as SCL:
   #_w1 := #alwaysON AND #State.Ready_For_Transfer;
   #_w2 := #_w1 AND #IN_Dose_Run;
   IF #_w2 THEN #State.Tank_Available := FALSE; END_IF;
   #Actuator.AV_Transfer := #_w2 AND #IN_Dose_Valve_Cmd AND #IN_Dose_LineOK;
   IF #_w1 AND #IN_FBAV_Outlet AND #IN_FBAV_Transfer AND #IN_Dose_LineOK AND #IN_FBP_Transfer THEN
       #State.Transfer_On_Prog := TRUE;
   END_IF;
   IF #alwaysON AND (NOT #State.Ready_For_Transfer OR (NOT #IN_Dose_Run AND NOT #IN_FBP_Transfer)) THEN
       #State.Transfer_On_Prog := FALSE;
   END_IF;
END_REGION

REGION Network 10: Command CIP
   RUNG wire#powerrail
      Contact( #alwaysON )
      wire#w1
      Contact( #State.Tank_LL )
      I_Contact( #"CIP Busy" )
      I_Contact( #State.Ready_For_Transfer )
      I_Contact( #State.Inloading )
      wire#w2
      I_Contact( #State.Line_inCIP )
      Coil( #State.Tank_CIP_Enable )
   END_RUNG
   RUNG wire#w2
      I_Contact( #State.Tank_inCIP )
      Coil( #State.Line_CIP_Enable )
   END_RUNG
   RUNG wire#w1
      Contact( #State.Tank_CIP_Enable )
      Contact( #Cmd.CIP_Tank )
      S_Coil( #State.Tank_inCIP )
   END_RUNG
   RUNG wire#w1
      I_Contact( #Cmd.CIP_Tank )
      R_Coil( #State.Tank_inCIP )
   END_RUNG
   RUNG wire#w1
      Contact( #State.Line_CIP_Enable )
      Contact( #Cmd.CIP_Line )
      S_Coil( #State.Line_inCIP )
   END_RUNG
   RUNG wire#w1
      I_Contact( #Cmd.CIP_Line )
      R_Coil( #State.Line_inCIP )
   END_RUNG
   RUNG wire#w1
      Contact( #State.Tank_inCIP )
      { S7_Templates := "SrcType := Real" } GE_Contact(in1 := #IN_LT01, in2 := #Param.CIP_Ret_ON_SP)
      S_Coil( #State.CIP_Return_On )
   END_RUNG
   RUNG wire#w1
      { S7_Templates := "SrcType := Real" } LE_Contact(in1 := #IN_LT01, in2 := #Param.CIP_Ret_OFF_SP)
      R_Coil( #State.CIP_Return_On )
   END_RUNG
   // the same network as SCL:
   #_w1 := #alwaysON AND #State.Tank_LL AND NOT #"CIP Busy" AND NOT #State.Ready_For_Transfer AND NOT #State.Inloading;
   #State.Tank_CIP_Enable := #_w1 AND NOT #State.Line_inCIP;
   #State.Line_CIP_Enable := #_w1 AND NOT #State.Tank_inCIP;
   IF #alwaysON AND #State.Tank_CIP_Enable AND #Cmd.CIP_Tank THEN #State.Tank_inCIP := TRUE; END_IF;
   IF #alwaysON AND NOT #Cmd.CIP_Tank THEN #State.Tank_inCIP := FALSE; END_IF;
   IF #alwaysON AND #State.Line_CIP_Enable AND #Cmd.CIP_Line THEN #State.Line_inCIP := TRUE; END_IF;
   IF #alwaysON AND NOT #Cmd.CIP_Line THEN #State.Line_inCIP := FALSE; END_IF;
   IF #alwaysON AND #State.Tank_inCIP AND (#IN_LT01 >= #Param.CIP_Ret_ON_SP) THEN
       #State.CIP_Return_On := TRUE;
   END_IF;
   IF #alwaysON AND (#IN_LT01 <= #Param.CIP_Ret_OFF_SP) THEN #State.CIP_Return_On := FALSE; END_IF;
END_REGION

REGION Network 11: Reset Command CIP
   RUNG wire#powerrail
      Contact( #alwaysON )
      Contact( #"CIP Complete" )
      P_Trig( #r.PosE2 )
      wire#w1
      R_Coil( #Cmd.CIP_Tank )
   END_RUNG
   RUNG wire#w1
      R_Coil( #Cmd.CIP_Line )
   END_RUNG
   // the same network as SCL:
   #_w1 := #alwaysON AND #"CIP Complete";
   #_w2 := #_w1 AND NOT #r.PosE2;   // rising edge
   #r.PosE2 := #_w1;
   IF #_w2 THEN
       #Cmd.CIP_Tank := FALSE;
       #Cmd.CIP_Line := FALSE;
   END_IF;
END_REGION

REGION Network 12: CIP Request and CIP Line Open
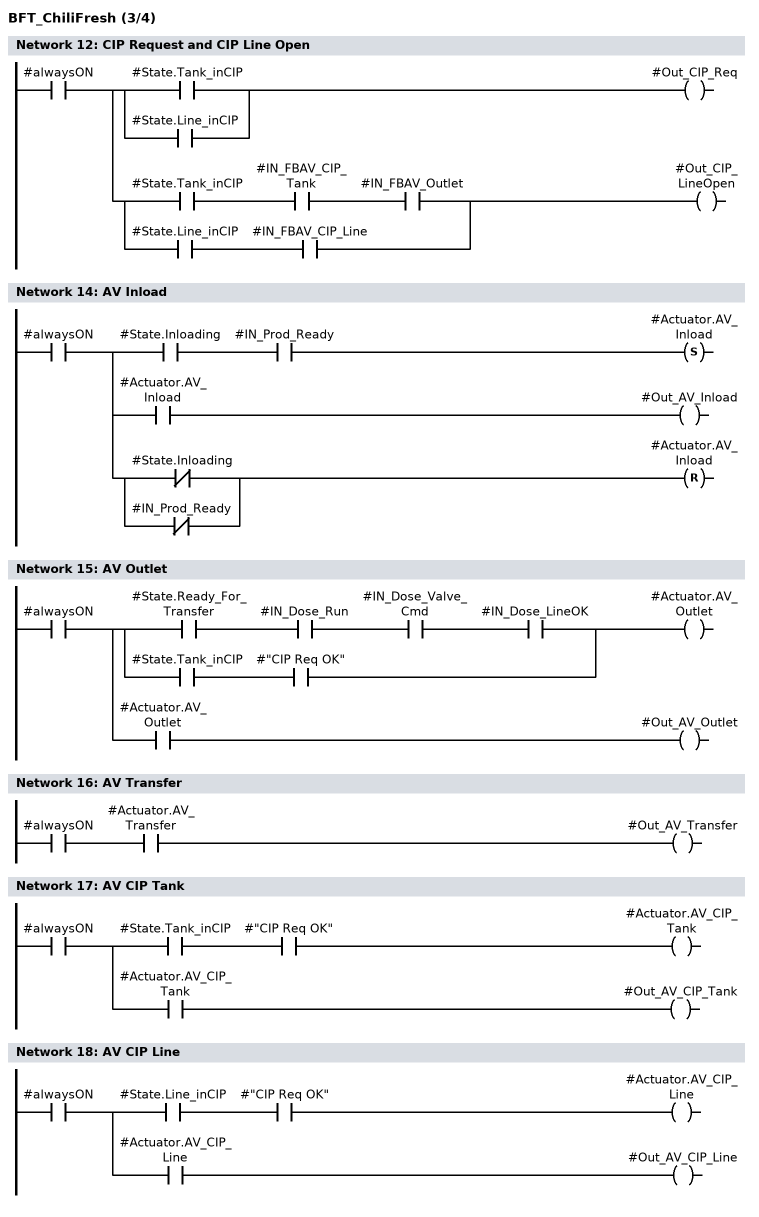
   RUNG wire#powerrail
      Contact( #alwaysON )
      wire#w1
      Contact( #State.Tank_inCIP )
      wire#w2
      Coil( #Out_CIP_Req )
   END_RUNG
   RUNG wire#w1
      Contact( #State.Line_inCIP )
   END_RUNG wire#w2
   RUNG wire#w1
      Contact( #State.Tank_inCIP )
      Contact( #IN_FBAV_CIP_Tank )
      Contact( #IN_FBAV_Outlet )
      wire#w3
      Coil( #Out_CIP_LineOpen )
   END_RUNG
   RUNG wire#w1
      Contact( #State.Line_inCIP )
      Contact( #IN_FBAV_CIP_Line )
   END_RUNG wire#w3
   // the same network as SCL:
   #Out_CIP_Req := #alwaysON AND (#State.Tank_inCIP OR #State.Line_inCIP);
   #Out_CIP_LineOpen := #alwaysON AND ((#State.Tank_inCIP AND #IN_FBAV_CIP_Tank AND #IN_FBAV_Outlet) OR (#State.Line_inCIP AND #IN_FBAV_CIP_Line));
END_REGION

REGION Network 14: AV Inload
   RUNG wire#powerrail
      Contact( #alwaysON )
      wire#w1
      Contact( #State.Inloading )
      Contact( #IN_Prod_Ready )
      S_Coil( #Actuator.AV_Inload )
   END_RUNG
   RUNG wire#w1
      Contact( #Actuator.AV_Inload )
      Coil( #Out_AV_Inload )
   END_RUNG
   RUNG wire#w1
      I_Contact( #State.Inloading )
      wire#w2
      R_Coil( #Actuator.AV_Inload )
   END_RUNG
   RUNG wire#w1
      I_Contact( #IN_Prod_Ready )
   END_RUNG wire#w2
   // the same network as SCL:
   IF #alwaysON AND #State.Inloading AND #IN_Prod_Ready THEN #Actuator.AV_Inload := TRUE; END_IF;
   #Out_AV_Inload := #alwaysON AND #Actuator.AV_Inload;
   IF #alwaysON AND (NOT #State.Inloading OR NOT #IN_Prod_Ready) THEN #Actuator.AV_Inload := FALSE; END_IF;
END_REGION

REGION Network 15: AV Outlet
   RUNG wire#powerrail
      Contact( #alwaysON )
      wire#w1
      Contact( #State.Ready_For_Transfer )
      Contact( #IN_Dose_Run )
      Contact( #IN_Dose_Valve_Cmd )
      Contact( #IN_Dose_LineOK )
      wire#w2
      Coil( #Actuator.AV_Outlet )
   END_RUNG
   RUNG wire#w1
      Contact( #State.Tank_inCIP )
      Contact( #"CIP Req OK" )
   END_RUNG wire#w2
   RUNG wire#w1
      Contact( #Actuator.AV_Outlet )
      Coil( #Out_AV_Outlet )
   END_RUNG
   // the same network as SCL:
   #Actuator.AV_Outlet := #alwaysON AND ((#State.Ready_For_Transfer AND #IN_Dose_Run AND #IN_Dose_Valve_Cmd AND #IN_Dose_LineOK) OR (#State.Tank_inCIP AND #"CIP Req OK"));
   #Out_AV_Outlet := #alwaysON AND #Actuator.AV_Outlet;
END_REGION

REGION Network 16: AV Transfer
   RUNG wire#powerrail
      Contact( #alwaysON )
      Contact( #Actuator.AV_Transfer )
      Coil( #Out_AV_Transfer )
   END_RUNG
   // the same network as SCL:
   #Out_AV_Transfer := #alwaysON AND #Actuator.AV_Transfer;
END_REGION

REGION Network 17: AV CIP Tank
   RUNG wire#powerrail
      Contact( #alwaysON )
      wire#w1
      Contact( #State.Tank_inCIP )
      Contact( #"CIP Req OK" )
      Coil( #Actuator.AV_CIP_Tank )
   END_RUNG
   RUNG wire#w1
      Contact( #Actuator.AV_CIP_Tank )
      Coil( #Out_AV_CIP_Tank )
   END_RUNG
   // the same network as SCL:
   #Actuator.AV_CIP_Tank := #alwaysON AND #State.Tank_inCIP AND #"CIP Req OK";
   #Out_AV_CIP_Tank := #alwaysON AND #Actuator.AV_CIP_Tank;
END_REGION

REGION Network 18: AV CIP Line
   RUNG wire#powerrail
      Contact( #alwaysON )
      wire#w1
      Contact( #State.Line_inCIP )
      Contact( #"CIP Req OK" )
      Coil( #Actuator.AV_CIP_Line )
   END_RUNG
   RUNG wire#w1
      Contact( #Actuator.AV_CIP_Line )
      Coil( #Out_AV_CIP_Line )
   END_RUNG
   // the same network as SCL:
   #Actuator.AV_CIP_Line := #alwaysON AND #State.Line_inCIP AND #"CIP Req OK";
   #Out_AV_CIP_Line := #alwaysON AND #Actuator.AV_CIP_Line;
END_REGION

REGION Network 20: Pump Inload
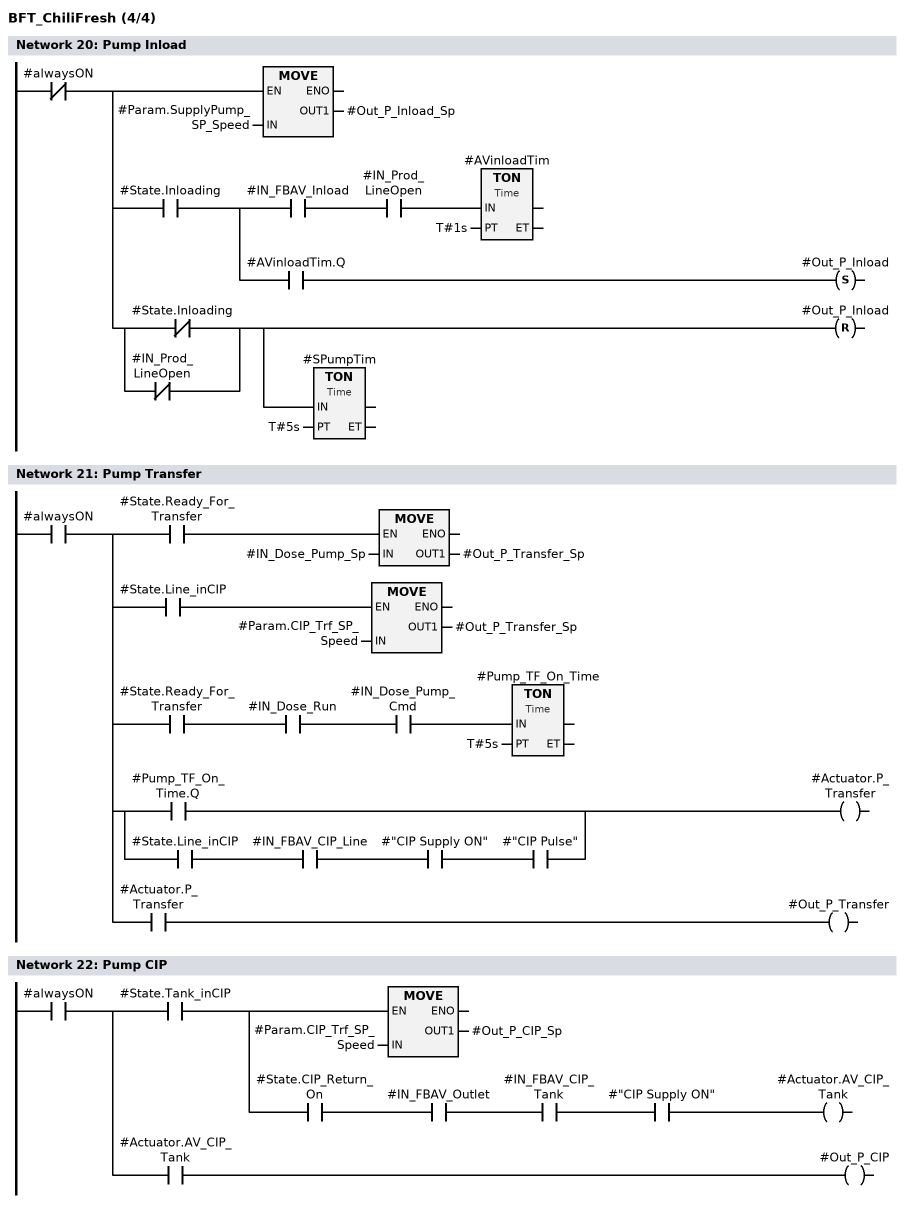
   RUNG wire#powerrail
      I_Contact( #alwaysON )
      wire#w1
      Move(in := #Param.SupplyPump_SP_Speed, out1 => #Out_P_Inload_Sp)
   END_RUNG
   RUNG wire#w1
      Contact( #State.Inloading )
      wire#w2
      Contact( #IN_FBAV_Inload )
      Contact( #IN_Prod_LineOpen )
      { S7_Templates := "time_type := Time" } #AVinloadTim.TON(pt := T#1s, et =>)
   END_RUNG
   RUNG wire#w2
      Contact( #AVinloadTim.Q )
      S_Coil( #Out_P_Inload )
   END_RUNG
   RUNG wire#w1
      I_Contact( #State.Inloading )
      wire#w3
      R_Coil( #Out_P_Inload )
   END_RUNG
   RUNG wire#w1
      I_Contact( #IN_Prod_LineOpen )
   END_RUNG wire#w3
   RUNG wire#w3
      { S7_Templates := "time_type := Time" } #SPumpTim.TON(pt := T#5s, et =>)
   END_RUNG
   // the same network as SCL:
   IF NOT #alwaysON THEN #Out_P_Inload_Sp := #Param.SupplyPump_SP_Speed; END_IF;
   #_w1 := NOT #alwaysON AND #State.Inloading;
   #AVinloadTim(IN := #_w1 AND #IN_FBAV_Inload AND #IN_Prod_LineOpen, PT := T#1s);   // TON
   IF #_w1 AND #AVinloadTim.Q THEN #Out_P_Inload := TRUE; END_IF;
   #_w2 := NOT #alwaysON AND (NOT #State.Inloading OR NOT #IN_Prod_LineOpen);
   IF #_w2 THEN #Out_P_Inload := FALSE; END_IF;
   #SPumpTim(IN := #_w2, PT := T#5s);   // TON
END_REGION

REGION Network 21: Pump Transfer
   RUNG wire#powerrail
      Contact( #alwaysON )
      wire#w1
      Contact( #State.Ready_For_Transfer )
      Move(in := #IN_Dose_Pump_Sp, out1 => #Out_P_Transfer_Sp)
   END_RUNG
   RUNG wire#w1
      Contact( #State.Line_inCIP )
      Move(in := #Param.CIP_Trf_SP_Speed, out1 => #Out_P_Transfer_Sp)
   END_RUNG
   RUNG wire#w1
      Contact( #State.Ready_For_Transfer )
      Contact( #IN_Dose_Run )
      Contact( #IN_Dose_Pump_Cmd )
      { S7_Templates := "time_type := Time" } #Pump_TF_On_Time.TON(pt := T#5s, et =>)
   END_RUNG
   RUNG wire#w1
      Contact( #Pump_TF_On_Time.Q )
      wire#w2
      Coil( #Actuator.P_Transfer )
   END_RUNG
   RUNG wire#w1
      Contact( #State.Line_inCIP )
      Contact( #IN_FBAV_CIP_Line )
      Contact( #"CIP Supply ON" )
      Contact( #"CIP Pulse" )
   END_RUNG wire#w2
   RUNG wire#w1
      Contact( #Actuator.P_Transfer )
      Coil( #Out_P_Transfer )
   END_RUNG
   // the same network as SCL:
   IF #alwaysON AND #State.Ready_For_Transfer THEN #Out_P_Transfer_Sp := #IN_Dose_Pump_Sp; END_IF;
   IF #alwaysON AND #State.Line_inCIP THEN #Out_P_Transfer_Sp := #Param.CIP_Trf_SP_Speed; END_IF;
   #Pump_TF_On_Time(IN := #alwaysON AND #State.Ready_For_Transfer AND #IN_Dose_Run AND #IN_Dose_Pump_Cmd,   // TON
                    PT := T#5s);
   #Actuator.P_Transfer := #alwaysON AND (#Pump_TF_On_Time.Q OR (#State.Line_inCIP AND #IN_FBAV_CIP_Line AND #"CIP Supply ON" AND #"CIP Pulse"));
   #Out_P_Transfer := #alwaysON AND #Actuator.P_Transfer;
END_REGION

REGION Network 22: Pump CIP
   RUNG wire#powerrail
      Contact( #alwaysON )
      wire#w1
      Contact( #State.Tank_inCIP )
      wire#w2
      Move(in := #Param.CIP_Trf_SP_Speed, out1 => #Out_P_CIP_Sp)
   END_RUNG
   RUNG wire#w2
      Contact( #State.CIP_Return_On )
      Contact( #IN_FBAV_Outlet )
      Contact( #IN_FBAV_CIP_Tank )
      Contact( #"CIP Supply ON" )
      Coil( #Actuator.AV_CIP_Tank )
   END_RUNG
   RUNG wire#w1
      Contact( #Actuator.AV_CIP_Tank )
      Coil( #Out_P_CIP )
   END_RUNG
   // the same network as SCL:
   #_w1 := #alwaysON AND #State.Tank_inCIP;
   IF #_w1 THEN #Out_P_CIP_Sp := #Param.CIP_Trf_SP_Speed; END_IF;
   #Actuator.AV_CIP_Tank := #_w1 AND #State.CIP_Return_On AND #IN_FBAV_Outlet AND #IN_FBAV_CIP_Tank AND #"CIP Supply ON";
   #Out_P_CIP := #alwaysON AND #Actuator.AV_CIP_Tank;
END_REGION
END_FUNCTION_BLOCK

FUNCTION_BLOCK "BFT_Garlic"   // FB362, LAD
{ S7_Optimized_Access := 'TRUE' }
VERSION : 0.1
// stored: AutoNumber false, IsIECCheckEnabled false, IsRetainMemResEnabled false, MemoryReserve 100, SetENOAutomatically false, UDAEnableTagReadback false
   VAR_INPUT
      IN_FBAV_Inload : Bool;
      IN_FBAV_Outlet : Bool;
      IN_FBAV_Transfer : Bool;
      IN_FBAV_CIP_Tank : Bool;
      IN_FBAV_CIP_Line : Bool;
      IN_FBP_Inload : Bool;
      IN_FBP_Inload_SP : Real;
      IN_FBP_Transfer : Bool;
      IN_FBP_Transfer_SP : Real;
      IN_FBP_CIP : Bool;
      IN_FBP_CIP_Sp : Real;
      IN_LT01 : Real;
      "LCS Start" : Bool;
      "LCS Stop" : Bool;
      "LCS EMS" : Bool;
      IN_Dose_Run : Bool;
      IN_Dose_Held : Bool;
      IN_Dose_Complete : Bool;
      IN_Dose_Header_1 : Bool;
      IN_Dose_Header_2 : Bool;
      IN_Dose_Valve_Cmd : Bool;
      IN_Dose_Pump_Cmd : Bool;
      IN_Dose_Pump_Sp : Real;
      IN_Dose_LineOK : Bool;
      "Inload Busy" : Bool;
      "CIP Pulse" : Bool;
      "CIP Supply ON" : Bool;
      "CIP Req OK" : Bool;
      "CIP Complete" : Bool;
      "CIP Busy" : Bool;
   END_VAR
   VAR_OUTPUT
      Out_AV_Inload : Bool;
      Out_AV_Outlet : Bool;
      Out_AV_Transfer : Bool;
      Out_AV_CIP_Tank : Bool;
      Out_AV_CIP_Line : Bool;
      Out_P_Inload : Bool;
      Out_P_Inload_Sp : Real;
      Out_P_Transfer : Bool;
      Out_P_Transfer_Sp : Real;
      Out_P_CIP : Bool;
      Out_P_CIP_Sp : Real;
      Out_XA : Bool;
      Out_XA_Speed : Real;
      Out_CIP_Req : Bool;
      Out_CIP_LineOpen : Bool;
   END_VAR
   VAR
      Cmd : Struct
         Inload : Bool;
         Ready_for_Tranfer : Bool;
         CIP_Tank : Bool;
         CIP_Line : Bool;
         Agitator_SpeedMode : Bool;
         Agitator_Mode : Bool;
         Agitator_Man_OnOff : Bool;
      END_STRUCT;
   END_VAR
   VAR RETAIN
      Param : Struct
         SP_Level_LL : Real := 10.0;
         SP_Level_ML : Real := 80.0;
         SP_Level_HL : Real := 100.0;
         SP_Level_Agi_ON1 : Real := 20.0;
         SP_Level_Agi_OFF1 : Real := 60.0;
         SP_Level_Agi_ON2 : Real := 62.0;
         SP_Level_Agi_OFF2 : Real := 80.0;
         SP_Level_Agi_ON3 : Real := 82.0;
         Agitator_SP_Speed : Real := 50.0;
         SupplyPump_SP_Speed : Real := 80.0;
         L_Hi_Lim : Real := 100.0;
         L_Lo_Lim : Real := 0.0;
         L_Hys : Real := 2.0;
         FlushingTime : DInt := 10000;
         CIP_Trf_SP_Speed : Real := 80.0;
         CIP_Ret_ON_SP : Real := 5.0;
         CIP_Ret_OFF_SP : Real;
      END_STRUCT;
   END_VAR
   VAR
      State : Struct   // Tank in loading state
         Tank_LL : Bool;
         Tank_ML : Bool;
         Tank_HL : Bool;
         Tank_inCIP : Bool;
         Tank_CIP_Enable : Bool;
         Line_inCIP : Bool;
         Line_CIP_Enable : Bool;
         CIP_Return_On : Bool;
         Inloading : Bool;
         Inload_Enable : Bool;
         Ready_For_Transfer : Bool;
         Ready_For_Transfer_Ena : Bool;
         Tank_Available : Bool;
         Transfer_On_Prog : Bool;
         L_Agi_ON1 : Bool;
         L_Agi_ON2 : Bool;
         L_Agi_ON3 : Bool;
      END_STRUCT;
      alwaysON : Bool;
      L_Hys_Abs : Real;
      Hys_Level_HL : Real;
      Hys_Level_ML : Real;
      Hys_Level_LL : Real;
      Hys_Level_Agi : Real;
      r : Struct
         PosE1 : Bool;
         PosE2 : Bool;
         PosE3 : Bool;
         PosE4 : Bool;
         PosE5 : Bool;
         PosE6 : Bool;
         PosE7 : Bool;
         PosE8 : Bool;
         PosE9 : Bool;
         PosE10 : Bool;
         PosE11 : Bool;
         PosE12 : Bool;
         PosE13 : Bool;
         PosE14 : Bool;
         PosE15 : Bool;
         PosE16 : Bool;
         PosE17 : Bool;
         PosE18 : Bool;
         PosE19 : Bool;
         PosE20 : Bool;
         PosE21 : Bool;
         PosE22 : Bool;
         PosE23 : Bool;
         PosE24 : Bool;
         PosE25 : Bool;
         PosE26 : Bool;
         PosE27 : Bool;
         PosE28 : Bool;
         PosE29 : Bool;
         PosE30 : Bool;
         PosE31 : Bool;
         PosE32 : Bool;
      END_STRUCT;
      Actuator : Struct
         AV_Inload : Bool;
         AV_Outlet : Bool;
         AV_Transfer : Bool;
         AV_CIP_Tank : Bool;
         AV_CIP_Line : Bool;
         P_Transfer : Bool;
         P_Inload : Bool;
         P_CIP : Bool;
         Agitator_level : Bool;
         LCS_OnOff : Bool;
      END_STRUCT;
      FlushingTim : TON_TIME;
      SPumpTim { S7_SetPoint := 'True'} : TON_TIME;
      AVinloadTim { S7_SetPoint := 'True'} : TON_TIME;
      L_AgiTim { S7_SetPoint := 'True'} : TON_TIME;
      Pump_TF_On_Time { S7_SetPoint := 'True'} : TON_TIME;
   END_VAR
   VAR_TEMP   // added for the SCL form of the ladder/FBD networks
      _w1 : Bool;
      _w2 : Bool;
   END_VAR
BEGIN

REGION Network 1: Always_ON
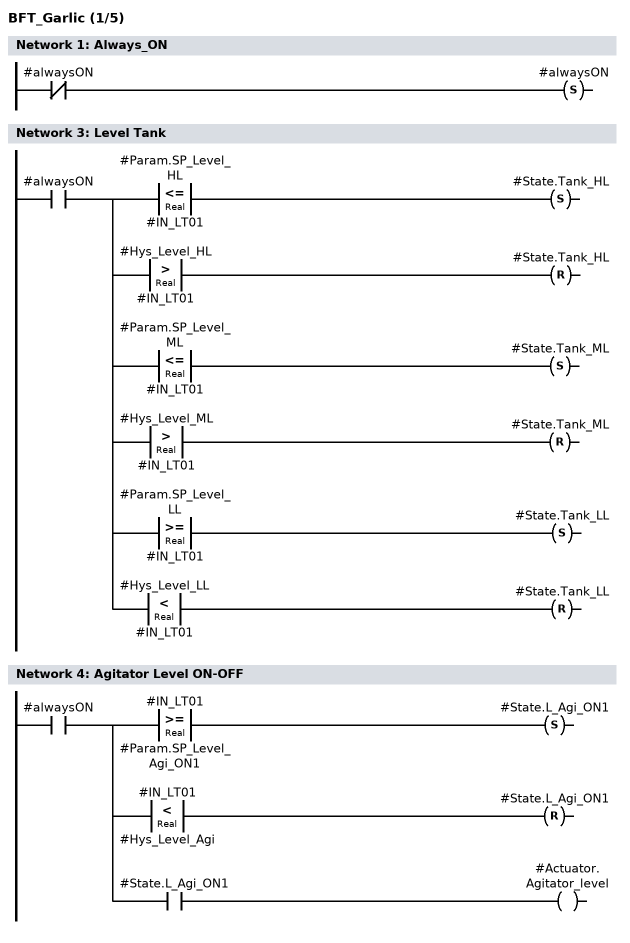
   RUNG wire#powerrail
      I_Contact( #alwaysON )
      S_Coil( #alwaysON )
   END_RUNG
   // the same network as SCL:
   IF NOT #alwaysON THEN #alwaysON := TRUE; END_IF;
END_REGION

NETWORK
TITLE = Hys Calculation
//Level Hys Absolute
      L     #Param.L_Hi_Lim;
      L     #Param.L_Lo_Lim;
      -R;
      L     100.0;
      /R;
      L     #Param.L_Hys;
      *R;
      T     #L_Hys_Abs;
//Tank High Level
      L     #Param.SP_Level_HL;
      L     #L_Hys_Abs;
      -R;
      T     #Hys_Level_HL;
//Tank Mid Level
      L     #Param.SP_Level_ML;
      L     #L_Hys_Abs;
      -R;
      T     #Hys_Level_ML;
//Tank Low Level
      L     #Param.SP_Level_LL;
      L     #L_Hys_Abs;
      +R;
      T     #Hys_Level_LL;
//Level Agi
      L     #Param.SP_Level_Agi_ON1;
      L     #L_Hys_Abs;
      -R;
      T     #Hys_Level_Agi;



REGION Network 3: Level Tank
   RUNG wire#powerrail
      Contact( #alwaysON )
      wire#w1
      { S7_Templates := "SrcType := Real" } LE_Contact(in1 := #Param.SP_Level_HL, in2 := #IN_LT01)
      S_Coil( #State.Tank_HL )
   END_RUNG
   RUNG wire#w1
      { S7_Templates := "SrcType := Real" } GT_Contact(in1 := #Hys_Level_HL, in2 := #IN_LT01)
      R_Coil( #State.Tank_HL )
   END_RUNG
   RUNG wire#w1
      { S7_Templates := "SrcType := Real" } LE_Contact(in1 := #Param.SP_Level_ML, in2 := #IN_LT01)
      S_Coil( #State.Tank_ML )
   END_RUNG
   RUNG wire#w1
      { S7_Templates := "SrcType := Real" } GT_Contact(in1 := #Hys_Level_ML, in2 := #IN_LT01)
      R_Coil( #State.Tank_ML )
   END_RUNG
   RUNG wire#w1
      { S7_Templates := "SrcType := Real" } GE_Contact(in1 := #Param.SP_Level_LL, in2 := #IN_LT01)
      S_Coil( #State.Tank_LL )
   END_RUNG
   RUNG wire#w1
      { S7_Templates := "SrcType := Real" } LT_Contact(in1 := #Hys_Level_LL, in2 := #IN_LT01)
      R_Coil( #State.Tank_LL )
   END_RUNG
   // the same network as SCL:
   IF #alwaysON AND (#Param.SP_Level_HL <= #IN_LT01) THEN #State.Tank_HL := TRUE; END_IF;
   IF #alwaysON AND (#Hys_Level_HL > #IN_LT01) THEN #State.Tank_HL := FALSE; END_IF;
   IF #alwaysON AND (#Param.SP_Level_ML <= #IN_LT01) THEN #State.Tank_ML := TRUE; END_IF;
   IF #alwaysON AND (#Hys_Level_ML > #IN_LT01) THEN #State.Tank_ML := FALSE; END_IF;
   IF #alwaysON AND (#Param.SP_Level_LL >= #IN_LT01) THEN #State.Tank_LL := TRUE; END_IF;
   IF #alwaysON AND (#Hys_Level_LL < #IN_LT01) THEN #State.Tank_LL := FALSE; END_IF;
END_REGION

REGION Network 4: Agitator Level ON-OFF
   RUNG wire#powerrail
      Contact( #alwaysON )
      wire#w1
      { S7_Templates := "SrcType := Real" } GE_Contact(in1 := #IN_LT01, in2 := #Param.SP_Level_Agi_ON1)
      S_Coil( #State.L_Agi_ON1 )
   END_RUNG
   RUNG wire#w1
      { S7_Templates := "SrcType := Real" } LT_Contact(in1 := #IN_LT01, in2 := #Hys_Level_Agi)
      R_Coil( #State.L_Agi_ON1 )
   END_RUNG
   RUNG wire#w1
      Contact( #State.L_Agi_ON1 )
      Coil( #Actuator.Agitator_level )
   END_RUNG
   // the same network as SCL:
   IF #alwaysON AND (#IN_LT01 >= #Param.SP_Level_Agi_ON1) THEN #State.L_Agi_ON1 := TRUE; END_IF;
   IF #alwaysON AND (#IN_LT01 < #Hys_Level_Agi) THEN #State.L_Agi_ON1 := FALSE; END_IF;
   #Actuator.Agitator_level := #alwaysON AND #State.L_Agi_ON1;
END_REGION

REGION Network 5: Agitator
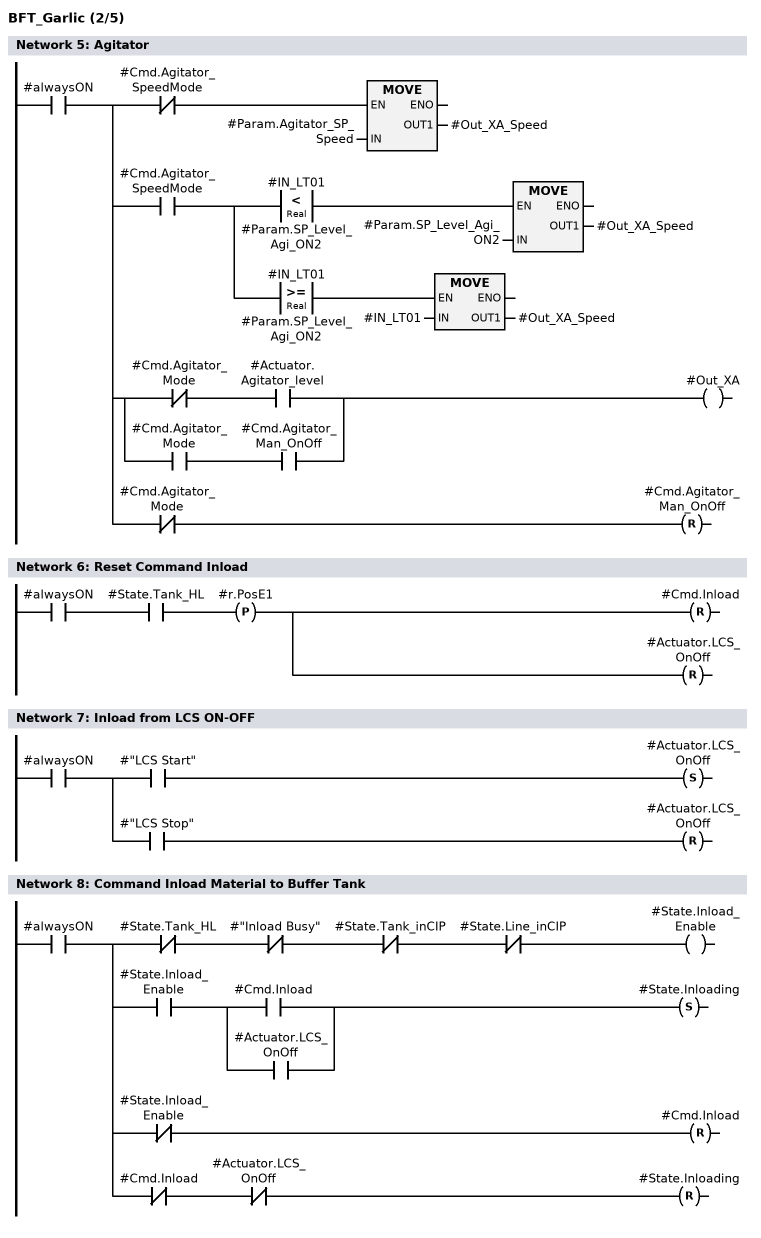
   RUNG wire#powerrail
      Contact( #alwaysON )
      wire#w1
      I_Contact( #Cmd.Agitator_SpeedMode )
      Move(in := #Param.Agitator_SP_Speed, out1 => #Out_XA_Speed)
   END_RUNG
   RUNG wire#w1
      Contact( #Cmd.Agitator_SpeedMode )
      wire#w2
      { S7_Templates := "SrcType := Real" } LT_Contact(in1 := #IN_LT01, in2 := #Param.SP_Level_Agi_ON2)
      Move(in := #Param.SP_Level_Agi_ON2, out1 => #Out_XA_Speed)
   END_RUNG
   RUNG wire#w2
      { S7_Templates := "SrcType := Real" } GE_Contact(in1 := #IN_LT01, in2 := #Param.SP_Level_Agi_ON2)
      Move(in := #IN_LT01, out1 => #Out_XA_Speed)
   END_RUNG
   RUNG wire#w1
      I_Contact( #Cmd.Agitator_Mode )
      Contact( #Actuator.Agitator_level )
      wire#w3
      Coil( #Out_XA )
   END_RUNG
   RUNG wire#w1
      Contact( #Cmd.Agitator_Mode )
      Contact( #Cmd.Agitator_Man_OnOff )
   END_RUNG wire#w3
   RUNG wire#w1
      I_Contact( #Cmd.Agitator_Mode )
      R_Coil( #Cmd.Agitator_Man_OnOff )
   END_RUNG
   // the same network as SCL:
   IF #alwaysON AND NOT #Cmd.Agitator_SpeedMode THEN #Out_XA_Speed := #Param.Agitator_SP_Speed; END_IF;
   #_w1 := #alwaysON AND #Cmd.Agitator_SpeedMode;
   IF #_w1 AND (#IN_LT01 < #Param.SP_Level_Agi_ON2) THEN #Out_XA_Speed := #Param.SP_Level_Agi_ON2; END_IF;
   IF #_w1 AND (#IN_LT01 >= #Param.SP_Level_Agi_ON2) THEN #Out_XA_Speed := #IN_LT01; END_IF;
   #Out_XA := #alwaysON AND ((NOT #Cmd.Agitator_Mode AND #Actuator.Agitator_level) OR (#Cmd.Agitator_Mode AND #Cmd.Agitator_Man_OnOff));
   IF #alwaysON AND NOT #Cmd.Agitator_Mode THEN #Cmd.Agitator_Man_OnOff := FALSE; END_IF;
END_REGION

REGION Network 6: Reset Command Inload
   RUNG wire#powerrail
      Contact( #alwaysON )
      Contact( #State.Tank_HL )
      P_Trig( #r.PosE1 )
      wire#w1
      R_Coil( #Cmd.Inload )
   END_RUNG
   RUNG wire#w1
      R_Coil( #Actuator.LCS_OnOff )
   END_RUNG
   // the same network as SCL:
   #_w1 := #alwaysON AND #State.Tank_HL;
   #_w2 := #_w1 AND NOT #r.PosE1;   // rising edge
   #r.PosE1 := #_w1;
   IF #_w2 THEN
       #Cmd.Inload := FALSE;
       #Actuator.LCS_OnOff := FALSE;
   END_IF;
END_REGION

REGION Network 7: Inload from LCS ON-OFF
   RUNG wire#powerrail
      Contact( #alwaysON )
      wire#w1
      Contact( #"LCS Start" )
      S_Coil( #Actuator.LCS_OnOff )
   END_RUNG
   RUNG wire#w1
      Contact( #"LCS Stop" )
      R_Coil( #Actuator.LCS_OnOff )
   END_RUNG
   // the same network as SCL:
   IF #alwaysON AND #"LCS Start" THEN #Actuator.LCS_OnOff := TRUE; END_IF;
   IF #alwaysON AND #"LCS Stop" THEN #Actuator.LCS_OnOff := FALSE; END_IF;
END_REGION

REGION Network 8: Command Inload Material to Buffer Tank
   RUNG wire#powerrail
      Contact( #alwaysON )
      wire#w1
      I_Contact( #State.Tank_HL )
      I_Contact( #"Inload Busy" )
      I_Contact( #State.Tank_inCIP )
      I_Contact( #State.Line_inCIP )
      Coil( #State.Inload_Enable )
   END_RUNG
   RUNG wire#w1
      Contact( #State.Inload_Enable )
      wire#w2
      Contact( #Cmd.Inload )
      wire#w3
      S_Coil( #State.Inloading )
   END_RUNG
   RUNG wire#w2
      Contact( #Actuator.LCS_OnOff )
   END_RUNG wire#w3
   RUNG wire#w1
      I_Contact( #State.Inload_Enable )
      R_Coil( #Cmd.Inload )
   END_RUNG
   RUNG wire#w1
      I_Contact( #Cmd.Inload )
      I_Contact( #Actuator.LCS_OnOff )
      R_Coil( #State.Inloading )
   END_RUNG
   // the same network as SCL:
   #State.Inload_Enable := #alwaysON AND NOT #State.Tank_HL AND NOT #"Inload Busy" AND NOT #State.Tank_inCIP AND NOT #State.Line_inCIP;
   IF #alwaysON AND #State.Inload_Enable AND (#Cmd.Inload OR #Actuator.LCS_OnOff) THEN
       #State.Inloading := TRUE;
   END_IF;
   IF #alwaysON AND NOT #State.Inload_Enable THEN #Cmd.Inload := FALSE; END_IF;
   IF #alwaysON AND NOT #Cmd.Inload AND NOT #Actuator.LCS_OnOff THEN #State.Inloading := FALSE; END_IF;
END_REGION

REGION Network 9: Tank Ready for Transfer to Blending
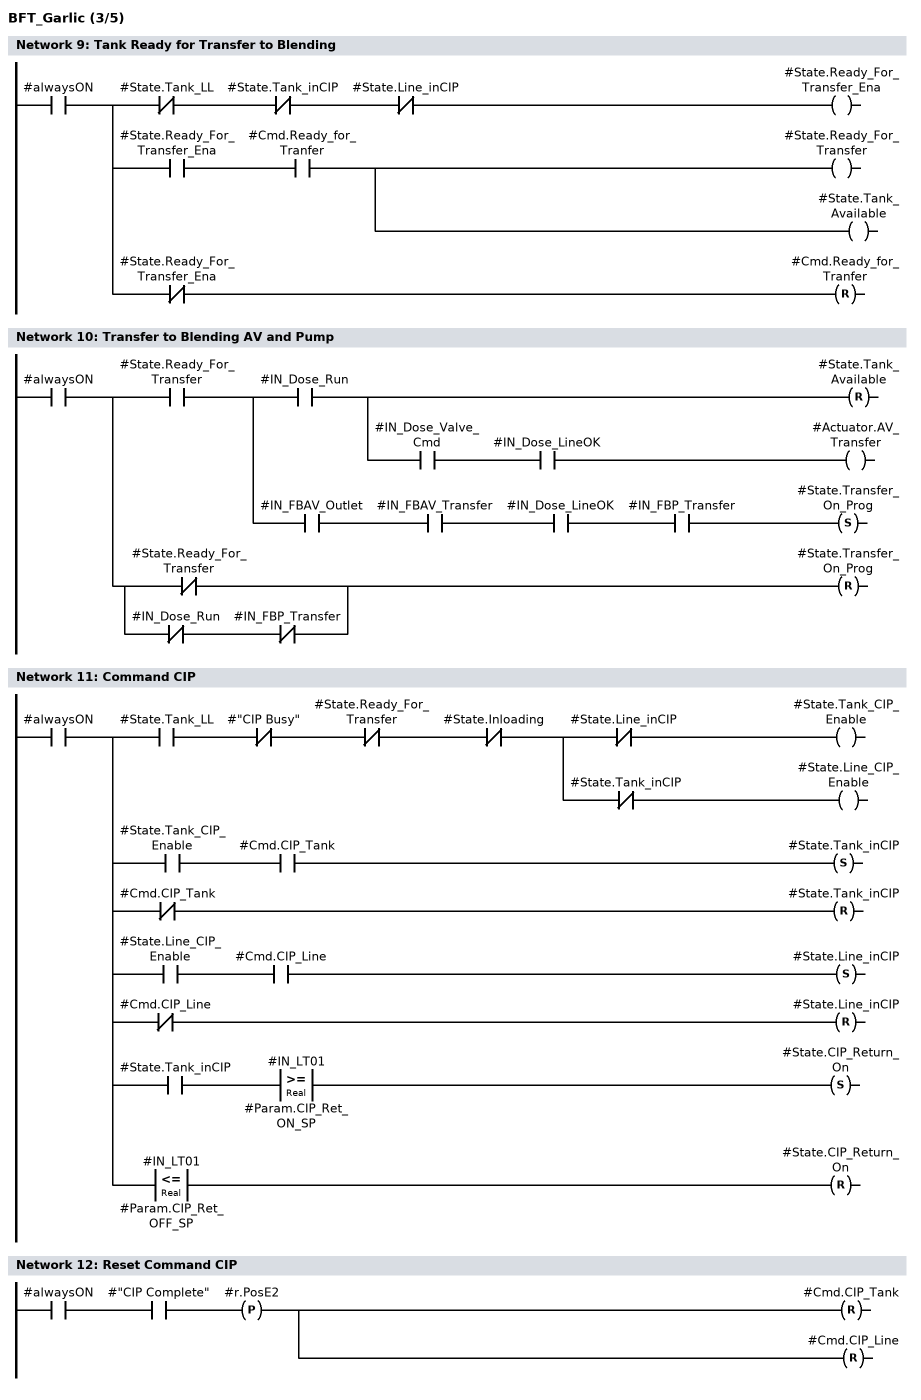
   RUNG wire#powerrail
      Contact( #alwaysON )
      wire#w1
      I_Contact( #State.Tank_LL )
      I_Contact( #State.Tank_inCIP )
      I_Contact( #State.Line_inCIP )
      Coil( #State.Ready_For_Transfer_Ena )
   END_RUNG
   RUNG wire#w1
      Contact( #State.Ready_For_Transfer_Ena )
      Contact( #Cmd.Ready_for_Tranfer )
      wire#w2
      Coil( #State.Ready_For_Transfer )
   END_RUNG
   RUNG wire#w2
      Coil( #State.Tank_Available )
   END_RUNG
   RUNG wire#w1
      I_Contact( #State.Ready_For_Transfer_Ena )
      R_Coil( #Cmd.Ready_for_Tranfer )
   END_RUNG
   // the same network as SCL:
   #State.Ready_For_Transfer_Ena := #alwaysON AND NOT #State.Tank_LL AND NOT #State.Tank_inCIP AND NOT #State.Line_inCIP;
   #State.Ready_For_Transfer := #alwaysON AND #State.Ready_For_Transfer_Ena AND #Cmd.Ready_for_Tranfer;
   #State.Tank_Available := #State.Ready_For_Transfer;
   IF #alwaysON AND NOT #State.Ready_For_Transfer_Ena THEN #Cmd.Ready_for_Tranfer := FALSE; END_IF;
END_REGION

REGION Network 10: Transfer to Blending AV and Pump
   RUNG wire#powerrail
      Contact( #alwaysON )
      wire#w1
      Contact( #State.Ready_For_Transfer )
      wire#w2
      Contact( #IN_Dose_Run )
      wire#w3
      R_Coil( #State.Tank_Available )
   END_RUNG
   RUNG wire#w3
      Contact( #IN_Dose_Valve_Cmd )
      Contact( #IN_Dose_LineOK )
      Coil( #Actuator.AV_Transfer )
   END_RUNG
   RUNG wire#w2
      Contact( #IN_FBAV_Outlet )
      Contact( #IN_FBAV_Transfer )
      Contact( #IN_Dose_LineOK )
      Contact( #IN_FBP_Transfer )
      S_Coil( #State.Transfer_On_Prog )
   END_RUNG
   RUNG wire#w1
      I_Contact( #State.Ready_For_Transfer )
      wire#w4
      R_Coil( #State.Transfer_On_Prog )
   END_RUNG
   RUNG wire#w1
      I_Contact( #IN_Dose_Run )
      I_Contact( #IN_FBP_Transfer )
   END_RUNG wire#w4
   // the same network as SCL:
   #_w1 := #alwaysON AND #State.Ready_For_Transfer;
   #_w2 := #_w1 AND #IN_Dose_Run;
   IF #_w2 THEN #State.Tank_Available := FALSE; END_IF;
   #Actuator.AV_Transfer := #_w2 AND #IN_Dose_Valve_Cmd AND #IN_Dose_LineOK;
   IF #_w1 AND #IN_FBAV_Outlet AND #IN_FBAV_Transfer AND #IN_Dose_LineOK AND #IN_FBP_Transfer THEN
       #State.Transfer_On_Prog := TRUE;
   END_IF;
   IF #alwaysON AND (NOT #State.Ready_For_Transfer OR (NOT #IN_Dose_Run AND NOT #IN_FBP_Transfer)) THEN
       #State.Transfer_On_Prog := FALSE;
   END_IF;
END_REGION

REGION Network 11: Command CIP
   RUNG wire#powerrail
      Contact( #alwaysON )
      wire#w1
      Contact( #State.Tank_LL )
      I_Contact( #"CIP Busy" )
      I_Contact( #State.Ready_For_Transfer )
      I_Contact( #State.Inloading )
      wire#w2
      I_Contact( #State.Line_inCIP )
      Coil( #State.Tank_CIP_Enable )
   END_RUNG
   RUNG wire#w2
      I_Contact( #State.Tank_inCIP )
      Coil( #State.Line_CIP_Enable )
   END_RUNG
   RUNG wire#w1
      Contact( #State.Tank_CIP_Enable )
      Contact( #Cmd.CIP_Tank )
      S_Coil( #State.Tank_inCIP )
   END_RUNG
   RUNG wire#w1
      I_Contact( #Cmd.CIP_Tank )
      R_Coil( #State.Tank_inCIP )
   END_RUNG
   RUNG wire#w1
      Contact( #State.Line_CIP_Enable )
      Contact( #Cmd.CIP_Line )
      S_Coil( #State.Line_inCIP )
   END_RUNG
   RUNG wire#w1
      I_Contact( #Cmd.CIP_Line )
      R_Coil( #State.Line_inCIP )
   END_RUNG
   RUNG wire#w1
      Contact( #State.Tank_inCIP )
      { S7_Templates := "SrcType := Real" } GE_Contact(in1 := #IN_LT01, in2 := #Param.CIP_Ret_ON_SP)
      S_Coil( #State.CIP_Return_On )
   END_RUNG
   RUNG wire#w1
      { S7_Templates := "SrcType := Real" } LE_Contact(in1 := #IN_LT01, in2 := #Param.CIP_Ret_OFF_SP)
      R_Coil( #State.CIP_Return_On )
   END_RUNG
   // the same network as SCL:
   #_w1 := #alwaysON AND #State.Tank_LL AND NOT #"CIP Busy" AND NOT #State.Ready_For_Transfer AND NOT #State.Inloading;
   #State.Tank_CIP_Enable := #_w1 AND NOT #State.Line_inCIP;
   #State.Line_CIP_Enable := #_w1 AND NOT #State.Tank_inCIP;
   IF #alwaysON AND #State.Tank_CIP_Enable AND #Cmd.CIP_Tank THEN #State.Tank_inCIP := TRUE; END_IF;
   IF #alwaysON AND NOT #Cmd.CIP_Tank THEN #State.Tank_inCIP := FALSE; END_IF;
   IF #alwaysON AND #State.Line_CIP_Enable AND #Cmd.CIP_Line THEN #State.Line_inCIP := TRUE; END_IF;
   IF #alwaysON AND NOT #Cmd.CIP_Line THEN #State.Line_inCIP := FALSE; END_IF;
   IF #alwaysON AND #State.Tank_inCIP AND (#IN_LT01 >= #Param.CIP_Ret_ON_SP) THEN
       #State.CIP_Return_On := TRUE;
   END_IF;
   IF #alwaysON AND (#IN_LT01 <= #Param.CIP_Ret_OFF_SP) THEN #State.CIP_Return_On := FALSE; END_IF;
END_REGION

REGION Network 12: Reset Command CIP
   RUNG wire#powerrail
      Contact( #alwaysON )
      Contact( #"CIP Complete" )
      P_Trig( #r.PosE2 )
      wire#w1
      R_Coil( #Cmd.CIP_Tank )
   END_RUNG
   RUNG wire#w1
      R_Coil( #Cmd.CIP_Line )
   END_RUNG
   // the same network as SCL:
   #_w1 := #alwaysON AND #"CIP Complete";
   #_w2 := #_w1 AND NOT #r.PosE2;   // rising edge
   #r.PosE2 := #_w1;
   IF #_w2 THEN
       #Cmd.CIP_Tank := FALSE;
       #Cmd.CIP_Line := FALSE;
   END_IF;
END_REGION

REGION Network 13: CIP Request and CIP Line Open
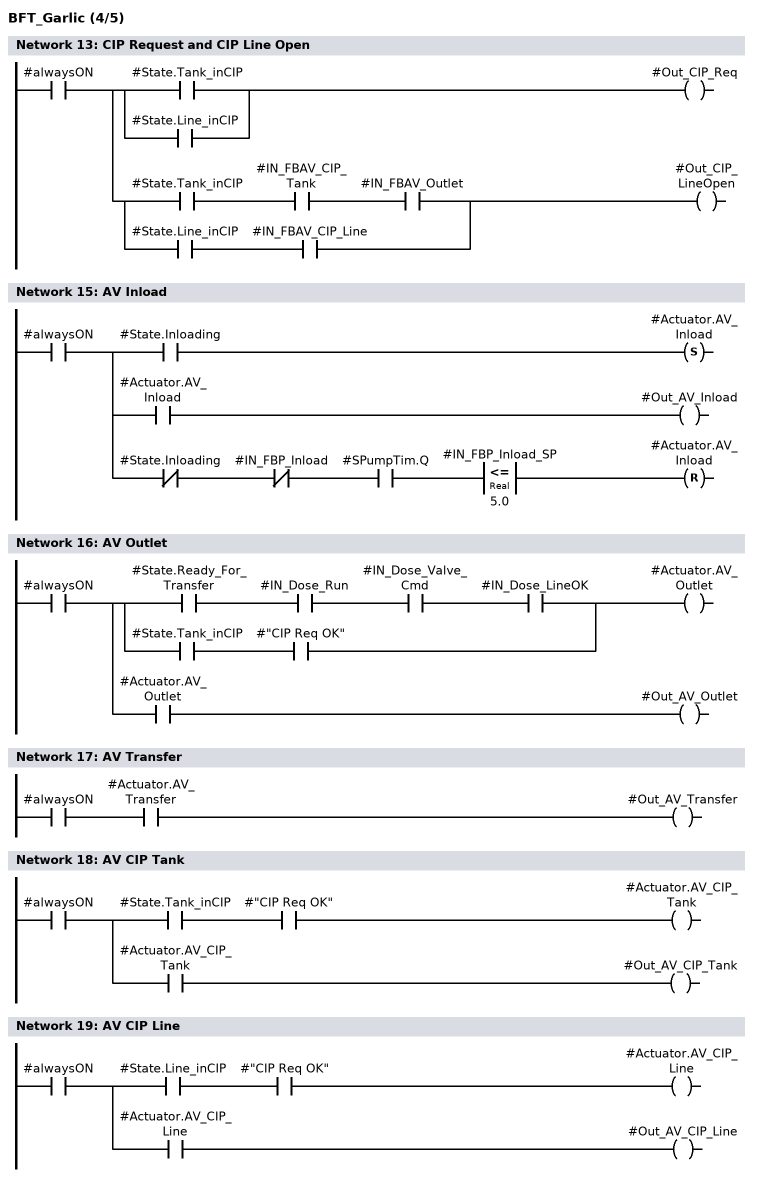
   RUNG wire#powerrail
      Contact( #alwaysON )
      wire#w1
      Contact( #State.Tank_inCIP )
      wire#w2
      Coil( #Out_CIP_Req )
   END_RUNG
   RUNG wire#w1
      Contact( #State.Line_inCIP )
   END_RUNG wire#w2
   RUNG wire#w1
      Contact( #State.Tank_inCIP )
      Contact( #IN_FBAV_CIP_Tank )
      Contact( #IN_FBAV_Outlet )
      wire#w3
      Coil( #Out_CIP_LineOpen )
   END_RUNG
   RUNG wire#w1
      Contact( #State.Line_inCIP )
      Contact( #IN_FBAV_CIP_Line )
   END_RUNG wire#w3
   // the same network as SCL:
   #Out_CIP_Req := #alwaysON AND (#State.Tank_inCIP OR #State.Line_inCIP);
   #Out_CIP_LineOpen := #alwaysON AND ((#State.Tank_inCIP AND #IN_FBAV_CIP_Tank AND #IN_FBAV_Outlet) OR (#State.Line_inCIP AND #IN_FBAV_CIP_Line));
END_REGION

REGION Network 15: AV Inload
   RUNG wire#powerrail
      Contact( #alwaysON )
      wire#w1
      Contact( #State.Inloading )
      S_Coil( #Actuator.AV_Inload )
   END_RUNG
   RUNG wire#w1
      Contact( #Actuator.AV_Inload )
      Coil( #Out_AV_Inload )
   END_RUNG
   RUNG wire#w1
      I_Contact( #State.Inloading )
      I_Contact( #IN_FBP_Inload )
      Contact( #SPumpTim.Q )
      { S7_Templates := "SrcType := Real" } LE_Contact(in1 := #IN_FBP_Inload_SP, in2 := 5.0)
      R_Coil( #Actuator.AV_Inload )
   END_RUNG
   // the same network as SCL:
   IF #alwaysON AND #State.Inloading THEN #Actuator.AV_Inload := TRUE; END_IF;
   #Out_AV_Inload := #alwaysON AND #Actuator.AV_Inload;
   IF #alwaysON AND NOT #State.Inloading AND NOT #IN_FBP_Inload AND #SPumpTim.Q AND (#IN_FBP_Inload_SP <= 5.0) THEN
       #Actuator.AV_Inload := FALSE;
   END_IF;
END_REGION

REGION Network 16: AV Outlet
   RUNG wire#powerrail
      Contact( #alwaysON )
      wire#w1
      Contact( #State.Ready_For_Transfer )
      Contact( #IN_Dose_Run )
      Contact( #IN_Dose_Valve_Cmd )
      Contact( #IN_Dose_LineOK )
      wire#w2
      Coil( #Actuator.AV_Outlet )
   END_RUNG
   RUNG wire#w1
      Contact( #State.Tank_inCIP )
      Contact( #"CIP Req OK" )
   END_RUNG wire#w2
   RUNG wire#w1
      Contact( #Actuator.AV_Outlet )
      Coil( #Out_AV_Outlet )
   END_RUNG
   // the same network as SCL:
   #Actuator.AV_Outlet := #alwaysON AND ((#State.Ready_For_Transfer AND #IN_Dose_Run AND #IN_Dose_Valve_Cmd AND #IN_Dose_LineOK) OR (#State.Tank_inCIP AND #"CIP Req OK"));
   #Out_AV_Outlet := #alwaysON AND #Actuator.AV_Outlet;
END_REGION

REGION Network 17: AV Transfer
   RUNG wire#powerrail
      Contact( #alwaysON )
      Contact( #Actuator.AV_Transfer )
      Coil( #Out_AV_Transfer )
   END_RUNG
   // the same network as SCL:
   #Out_AV_Transfer := #alwaysON AND #Actuator.AV_Transfer;
END_REGION

REGION Network 18: AV CIP Tank
   RUNG wire#powerrail
      Contact( #alwaysON )
      wire#w1
      Contact( #State.Tank_inCIP )
      Contact( #"CIP Req OK" )
      Coil( #Actuator.AV_CIP_Tank )
   END_RUNG
   RUNG wire#w1
      Contact( #Actuator.AV_CIP_Tank )
      Coil( #Out_AV_CIP_Tank )
   END_RUNG
   // the same network as SCL:
   #Actuator.AV_CIP_Tank := #alwaysON AND #State.Tank_inCIP AND #"CIP Req OK";
   #Out_AV_CIP_Tank := #alwaysON AND #Actuator.AV_CIP_Tank;
END_REGION

REGION Network 19: AV CIP Line
   RUNG wire#powerrail
      Contact( #alwaysON )
      wire#w1
      Contact( #State.Line_inCIP )
      Contact( #"CIP Req OK" )
      Coil( #Actuator.AV_CIP_Line )
   END_RUNG
   RUNG wire#w1
      Contact( #Actuator.AV_CIP_Line )
      Coil( #Out_AV_CIP_Line )
   END_RUNG
   // the same network as SCL:
   #Actuator.AV_CIP_Line := #alwaysON AND #State.Line_inCIP AND #"CIP Req OK";
   #Out_AV_CIP_Line := #alwaysON AND #Actuator.AV_CIP_Line;
END_REGION

REGION Network 21: Pump Inload
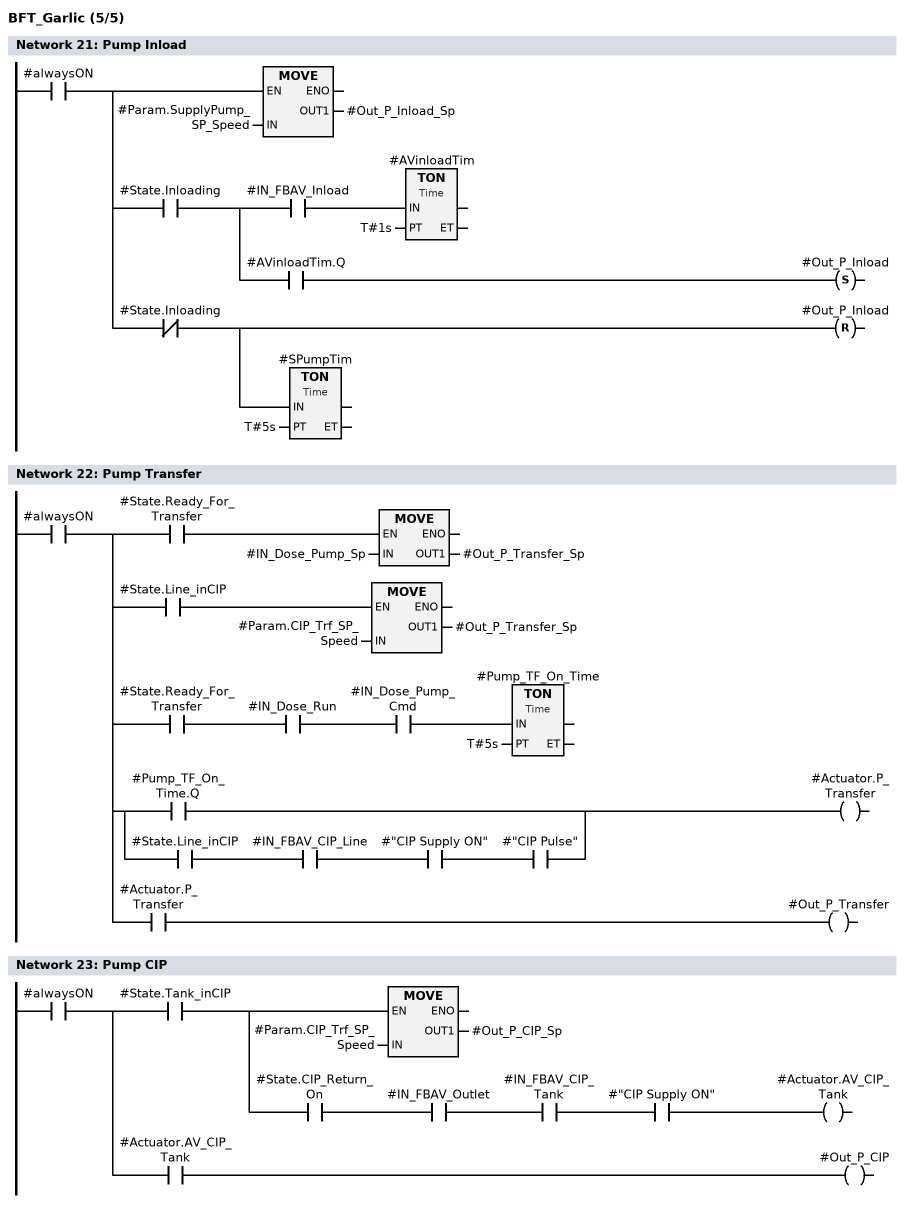
   RUNG wire#powerrail
      Contact( #alwaysON )
      wire#w1
      Move(in := #Param.SupplyPump_SP_Speed, out1 => #Out_P_Inload_Sp)
   END_RUNG
   RUNG wire#w1
      Contact( #State.Inloading )
      wire#w2
      Contact( #IN_FBAV_Inload )
      { S7_Templates := "time_type := Time" } #AVinloadTim.TON(pt := T#1s, et =>)
   END_RUNG
   RUNG wire#w2
      Contact( #AVinloadTim.Q )
      S_Coil( #Out_P_Inload )
   END_RUNG
   RUNG wire#w1
      I_Contact( #State.Inloading )
      wire#w3
      R_Coil( #Out_P_Inload )
   END_RUNG
   RUNG wire#w3
      { S7_Templates := "time_type := Time" } #SPumpTim.TON(pt := T#5s, et =>)
   END_RUNG
   // the same network as SCL:
   IF #alwaysON THEN #Out_P_Inload_Sp := #Param.SupplyPump_SP_Speed; END_IF;
   #_w1 := #alwaysON AND #State.Inloading;
   #AVinloadTim(IN := #_w1 AND #IN_FBAV_Inload, PT := T#1s);   // TON
   IF #_w1 AND #AVinloadTim.Q THEN #Out_P_Inload := TRUE; END_IF;
   #_w2 := #alwaysON AND NOT #State.Inloading;
   IF #_w2 THEN #Out_P_Inload := FALSE; END_IF;
   #SPumpTim(IN := #_w2, PT := T#5s);   // TON
END_REGION

REGION Network 22: Pump Transfer
   RUNG wire#powerrail
      Contact( #alwaysON )
      wire#w1
      Contact( #State.Ready_For_Transfer )
      Move(in := #IN_Dose_Pump_Sp, out1 => #Out_P_Transfer_Sp)
   END_RUNG
   RUNG wire#w1
      Contact( #State.Line_inCIP )
      Move(in := #Param.CIP_Trf_SP_Speed, out1 => #Out_P_Transfer_Sp)
   END_RUNG
   RUNG wire#w1
      Contact( #State.Ready_For_Transfer )
      Contact( #IN_Dose_Run )
      Contact( #IN_Dose_Pump_Cmd )
      { S7_Templates := "time_type := Time" } #Pump_TF_On_Time.TON(pt := T#5s, et =>)
   END_RUNG
   RUNG wire#w1
      Contact( #Pump_TF_On_Time.Q )
      wire#w2
      Coil( #Actuator.P_Transfer )
   END_RUNG
   RUNG wire#w1
      Contact( #State.Line_inCIP )
      Contact( #IN_FBAV_CIP_Line )
      Contact( #"CIP Supply ON" )
      Contact( #"CIP Pulse" )
   END_RUNG wire#w2
   RUNG wire#w1
      Contact( #Actuator.P_Transfer )
      Coil( #Out_P_Transfer )
   END_RUNG
   // the same network as SCL:
   IF #alwaysON AND #State.Ready_For_Transfer THEN #Out_P_Transfer_Sp := #IN_Dose_Pump_Sp; END_IF;
   IF #alwaysON AND #State.Line_inCIP THEN #Out_P_Transfer_Sp := #Param.CIP_Trf_SP_Speed; END_IF;
   #Pump_TF_On_Time(IN := #alwaysON AND #State.Ready_For_Transfer AND #IN_Dose_Run AND #IN_Dose_Pump_Cmd,   // TON
                    PT := T#5s);
   #Actuator.P_Transfer := #alwaysON AND (#Pump_TF_On_Time.Q OR (#State.Line_inCIP AND #IN_FBAV_CIP_Line AND #"CIP Supply ON" AND #"CIP Pulse"));
   #Out_P_Transfer := #alwaysON AND #Actuator.P_Transfer;
END_REGION

REGION Network 23: Pump CIP
   RUNG wire#powerrail
      Contact( #alwaysON )
      wire#w1
      Contact( #State.Tank_inCIP )
      wire#w2
      Move(in := #Param.CIP_Trf_SP_Speed, out1 => #Out_P_CIP_Sp)
   END_RUNG
   RUNG wire#w2
      Contact( #State.CIP_Return_On )
      Contact( #IN_FBAV_Outlet )
      Contact( #IN_FBAV_CIP_Tank )
      Contact( #"CIP Supply ON" )
      Coil( #Actuator.AV_CIP_Tank )
   END_RUNG
   RUNG wire#w1
      Contact( #Actuator.AV_CIP_Tank )
      Coil( #Out_P_CIP )
   END_RUNG
   // the same network as SCL:
   #_w1 := #alwaysON AND #State.Tank_inCIP;
   IF #_w1 THEN #Out_P_CIP_Sp := #Param.CIP_Trf_SP_Speed; END_IF;
   #Actuator.AV_CIP_Tank := #_w1 AND #State.CIP_Return_On AND #IN_FBAV_Outlet AND #IN_FBAV_CIP_Tank AND #"CIP Supply ON";
   #Out_P_CIP := #alwaysON AND #Actuator.AV_CIP_Tank;
END_REGION
END_FUNCTION_BLOCK

FUNCTION_BLOCK "BFT_Vinegar"   // FB363, LAD
{ S7_Optimized_Access := 'TRUE' }
VERSION : 0.1
// stored: AutoNumber false, IsIECCheckEnabled false, IsRetainMemResEnabled false, MemoryReserve 100, SetENOAutomatically false, UDAEnableTagReadback false
   VAR_INPUT
      IN_FBAV_Inload : Bool;
      IN_FBAV_Outlet : Bool;
      IN_FBAV_Transfer : Bool;
      IN_FBAV_CIP_Tank : Bool;
      IN_FBAV_CIP_Line : Bool;
      IN_FBP_Inload : Bool;
      IN_FBP_Inload_SP : Real;
      IN_FBP_Transfer : Bool;
      IN_FBP_Transfer_SP : Real;
      IN_FBP_CIP : Bool;
      IN_FBP_CIP_Sp : Real;
      IN_LT01 : Real;
      "LCS Start" : Bool;
      "LCS Stop" : Bool;
      "LCS EMS" : Bool;
      IN_Dose_Run : Bool;
      IN_Dose_Held : Bool;
      IN_Dose_Complete : Bool;
      IN_Dose_Valve_Cmd : Bool;
      IN_Dose_Pump_Cmd : Bool;
      IN_Dose_Pump_Sp : Real;
      IN_Dose_LineOK : Bool;
      "Inload Busy" : Bool;
      "CIP Pulse" : Bool;
      "CIP Supply ON" : Bool;
      "CIP Req OK" : Bool;
      "CIP Complete" : Bool;
      "CIP Busy" : Bool;
   END_VAR
   VAR_OUTPUT
      Out_AV_Inload : Bool;
      Out_AV_Outlet : Bool;
      Out_AV_Transfer : Bool;
      Out_AV_CIP_Tank : Bool;
      Out_AV_CIP_Line : Bool;
      Out_P_Inload : Bool;
      Out_P_Inload_Sp : Real;
      Out_P_Transfer : Bool;
      Out_P_Transfer_Sp : Real;
      Out_P_CIP : Bool;
      Out_P_CIP_Sp : Real;
      Out_CIP_Req : Bool;
      Out_CIP_LineOpen : Bool;
   END_VAR
   VAR
      Cmd : Struct
         Inload : Bool;
         Ready_for_Tranfer : Bool;
         CIP_Tank : Bool;
         CIP_Line : Bool;
      END_STRUCT;
   END_VAR
   VAR RETAIN
      Param : Struct
         SP_Level_LL : Real := 10.0;
         SP_Level_ML : Real := 80.0;
         SP_Level_HL : Real := 100.0;
         SupplyPump_SP_Speed : Real := 80.0;
         L_Hi_Lim : Real := 100.0;
         L_Lo_Lim : Real := 0.0;
         L_Hys : Real := 2.0;
         FlushingTime : DInt := 10000;
         CIP_Trf_SP_Speed : Real := 80.0;
         CIP_Ret_ON_SP : Real := 5.0;
         CIP_Ret_OFF_SP : Real;
      END_STRUCT;
   END_VAR
   VAR
      State : Struct   // Tank in loading state
         Tank_LL : Bool;
         Tank_ML : Bool;
         Tank_HL : Bool;
         Tank_inCIP : Bool;
         Tank_CIP_Enable : Bool;
         Line_inCIP : Bool;
         Line_CIP_Enable : Bool;
         CIP_Return_On : Bool;
         Inloading : Bool;
         Inload_Enable : Bool;
         Ready_For_Transfer : Bool;
         Ready_For_Transfer_Ena : Bool;
         Tank_Available : Bool;
         Transfer_On_Prog : Bool;
      END_STRUCT;
      alwaysON : Bool;
      L_Hys_Abs : Real;
      Hys_Level_HL : Real;
      Hys_Level_ML : Real;
      Hys_Level_LL : Real;
      r : Struct
         PosE1 : Bool;
         PosE2 : Bool;
         PosE3 : Bool;
         PosE4 : Bool;
         PosE5 : Bool;
         PosE6 : Bool;
         PosE7 : Bool;
         PosE8 : Bool;
         PosE9 : Bool;
         PosE10 : Bool;
         PosE11 : Bool;
         PosE12 : Bool;
         PosE13 : Bool;
         PosE14 : Bool;
         PosE15 : Bool;
         PosE16 : Bool;
         PosE17 : Bool;
         PosE18 : Bool;
         PosE19 : Bool;
         PosE20 : Bool;
         PosE21 : Bool;
         PosE22 : Bool;
         PosE23 : Bool;
         PosE24 : Bool;
         PosE25 : Bool;
         PosE26 : Bool;
         PosE27 : Bool;
         PosE28 : Bool;
         PosE29 : Bool;
         PosE30 : Bool;
         PosE31 : Bool;
         PosE32 : Bool;
      END_STRUCT;
      Actuator : Struct
         AV_Inload : Bool;
         AV_Outlet : Bool;
         AV_Transfer : Bool;
         AV_CIP_Tank : Bool;
         AV_CIP_Line : Bool;
         P_Transfer : Bool;
         P_Inload : Bool;
         P_CIP : Bool;
         LCS_OnOff : Bool;
      END_STRUCT;
      FlushingTim : TON_TIME;
      SPumpTim { S7_SetPoint := 'True'} : TON_TIME;
      AVinloadTim { S7_SetPoint := 'True'} : TON_TIME;
      Pump_TF_On_Time { S7_SetPoint := 'True'} : TON_TIME;
   END_VAR
   VAR_TEMP   // added for the SCL form of the ladder/FBD networks
      _w1 : Bool;
      _w2 : Bool;
   END_VAR
BEGIN

REGION Network 1: Always_ON
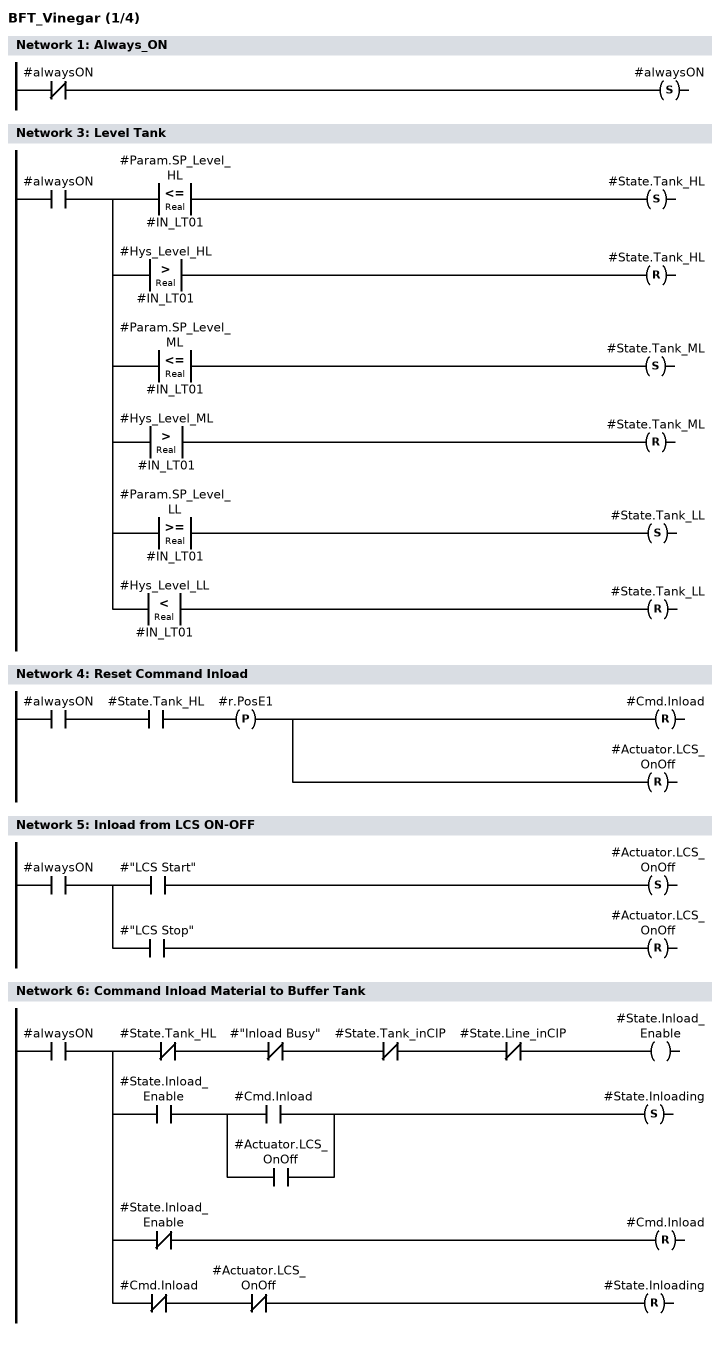
   RUNG wire#powerrail
      I_Contact( #alwaysON )
      S_Coil( #alwaysON )
   END_RUNG
   // the same network as SCL:
   IF NOT #alwaysON THEN #alwaysON := TRUE; END_IF;
END_REGION

